LIN {X 0,Y 305.438,Z 295.055,A -85,B 0,C 180,E1 -15812.6,E2 -15812.6} C_VEL
LIN {X 0,Y 305.444,Z 295.06,A -85,B 0,C 180,E1 -15815.533,E2 -15815.533} C_VEL
LIN {X 0,Y 305.473,Z 295.058,A -85,B 0,C 180,E1 -15819.812,E2 -15819.812} C_VEL
LIN {X 0,Y 305.509,Z 295.056,A -85,B 0,C 180,E1 -15823.975,E2 -15823.975} C_VEL
LIN {X 0,Y 305.569,Z 295.038,A -85,B 0,C 180,E1 -15826.703,E2 -15826.703} C_VEL
LIN {X 0,Y 305.751,Z 295.012,A -85,B 0,C 180,E1 -15831.261,E2 -15831.261} C_VEL
LIN {X 0,Y 305.782,Z 295.02,A -85,B 0,C 180,E1 -15833.401,E2 -15833.401} C_VEL
LIN {X 0,Y 305.869,Z 295.005,A -85,B 0,C 180,E1 -15837.366,E2 -15837.366} C_VEL
LIN {X 0,Y 305.914,Z 294.996,A -85,B 0,C 180,E1 -15840,E2 -15840} C_VEL
LIN {X 0,Y 305.856,Z 295.009,A -85,B 0,C 180,E1 -15842.634,E2 -15842.634} C_VEL
LIN {X 0,Y 305.785,Z 295.01,A -85,B 0,C 180,E1 -15846.599,E2 -15846.599} C_VEL
LIN {X 0,Y 305.692,Z 295.03,A -85,B 0,C 180,E1 -15849.261,E2 -15849.261} C_VEL
LIN {X 0,Y 305.588,Z 295.045,A -85,B 0,C 180,E1 -15853.296,E2 -15853.296} C_VEL
LIN {X 0,Y 305.592,Z 295.037,A -85,B 0,C 180,E1 -15856.02,E2 -15856.02} C_VEL
LIN {X 0,Y 305.575,Z 295.039,A -85,B 0,C 180,E1 -15859.445,E2 -15859.445} C_VEL
LIN {X 0,Y 305.484,Z 295.047,A -85,B 0,C 180,E1 -15863.039,E2 -15863.039} C_VEL
LIN {X 0,Y 305.469,Z 295.029,A -85,B 0,C 180,E1 -15866.198,E2 -15866.198} C_VEL
LIN {X 0,Y 305.456,Z 295.061,A -85,B 0,C 180,E1 -15869.037,E2 -15869.037} C_VEL
LIN {X 0,Y 305.434,Z 295.035,A -85,B 0,C 180,E1 -15871.953,E2 -15871.953} C_VEL
LIN {X 0,Y 305.461,Z 295.061,A -85,B 0,C 180,E1 -15875.113,E2 -15875.113} C_VEL
LIN {X 0,Y 305.438,Z 295.047,A -85,B 0,C 180,E1 -15878.527,E2 -15878.527} C_VEL
LIN {X 0,Y 305.453,Z 295.061,A -85,B 0,C 180,E1 -15882.586,E2 -15882.586} C_VEL
LIN {X 0,Y 305.445,Z 295.147,A -85,B 0,C 180,E1 -15886.483,E2 -15886.483} C_VEL
LIN {X 0,Y 308.84,Z 306.244,A -85,B 0,C 180,E1 -15890.054,E2 -15890.054} C_VEL
LIN {X 0,Y 310.401,Z 311.623,A -85,B 0,C 180,E1 -15891.632,E2 -15891.632} C_VEL
LIN {X 0,Y 319.441,Z 329.134,A -85,B 0,C 180,E1 -15893.374,E2 -15893.374} C_VEL
LIN {X 0,Y 328.319,Z 348.755,A -85,B 0,C 180,E1 -15895.02,E2 -15895.02} C_VEL
LIN {X 0,Y 331.337,Z 366.984,A -85,B 0,C 180,E1 -15895.849,E2 -15895.849} C_VEL
LIN {X 0,Y 328.248,Z 458.224,A -85,B 0,C 180,E1 -15897.82,E2 -15897.82} C_VEL
LIN {X 0,Y 327.28,Z 480.74,A -85,B 0,C 180,E1 -15898.348,E2 -15898.348} C_VEL
LIN {X 0,Y 325.993,Z 496.154,A -85,B 0,C 180,E1 -15898.932,E2 -15898.932} C_VEL
LIN {X 0,Y 324.176,Z 511.053,A -85,B 0,C 180,E1 -15899.732,E2 -15899.732} C_VEL
LIN {X 0,Y 322.054,Z 525.725,A -85,B 0,C 180,E1 -15900.797,E2 -15900.797} C_VEL
LIN {X 0,Y 319.866,Z 538.691,A -85,B 0,C 180,E1 -15901.989,E2 -15901.989} C_VEL
LIN {X 0,Y 317.244,Z 552.138,A -85,B 0,C 180,E1 -15903.524,E2 -15903.524} C_VEL
LIN {X 0,Y 314.639,Z 564.393,A -85,B 0,C 180,E1 -15905.241,E2 -15905.241} C_VEL
LIN {X 0,Y 312.196,Z 575.594,A -85,B 0,C 180,E1 -15907.15,E2 -15907.15} C_VEL
LIN {X 0,Y 310.158,Z 585.029,A -85,B 0,C 180,E1 -15909.092,E2 -15909.092} C_VEL
LIN {X 0,Y 308.094,Z 594.317,A -85,B 0,C 180,E1 -15911.377,E2 -15911.377} C_VEL
LIN {X 0,Y 306.236,Z 603.068,A -85,B 0,C 180,E1 -15914.015,E2 -15914.015} C_VEL
LIN {X 0,Y 304.974,Z 610.103,A -85,B 0,C 180,E1 -15916.677,E2 -15916.677} C_VEL
LIN {X 0,Y 304.129,Z 615.64,A -85,B 0,C 180,E1 -15919.347,E2 -15919.347} C_VEL
LIN {X 0,Y 303.744,Z 619.836,A -85,B 0,C 180,E1 -15922.021,E2 -15922.021} C_VEL
LIN {X 0,Y 303.616,Z 622.781,A -85,B 0,C 180,E1 -15924.688,E2 -15924.688} C_VEL
LIN {X 0,Y 303.621,Z 624.54,A -85,B 0,C 180,E1 -15927.347,E2 -15927.347} C_VEL
LIN {X 0,Y 303.667,Z 625.142,A -85,B 0,C 180,E1 -15930.001,E2 -15930.001} C_VEL
LIN {X 0,Y 303.621,Z 624.53,A -85,B 0,C 180,E1 -15932.654,E2 -15932.654} C_VEL
LIN {X 0,Y 303.624,Z 622.559,A -85,B 0,C 180,E1 -15935.545,E2 -15935.545} C_VEL
LIN {X 0,Y 303.743,Z 619.805,A -85,B 0,C 180,E1 -15937.981,E2 -15937.981} C_VEL
LIN {X 0,Y 304.118,Z 615.604,A -85,B 0,C 180,E1 -15940.655,E2 -15940.655} C_VEL
LIN {X 0,Y 304.975,Z 610.051,A -85,B 0,C 180,E1 -15943.324,E2 -15943.324} C_VEL
LIN {X 0,Y 306.237,Z 602.995,A -85,B 0,C 180,E1 -15945.986,E2 -15945.986} C_VEL
LIN {X 0,Y 308.037,Z 594.228,A -85,B 0,C 180,E1 -15948.628,E2 -15948.628} C_VEL
LIN {X 0,Y 310.17,Z 584.929,A -85,B 0,C 180,E1 -15950.909,E2 -15950.909} C_VEL
LIN {X 0,Y 312.217,Z 575.478,A -85,B 0,C 180,E1 -15952.849,E2 -15952.849} C_VEL
LIN {X 0,Y 314.826,Z 563.229,A -85,B 0,C 180,E1 -15954.921,E2 -15954.921} C_VEL
LIN {X 0,Y 317.458,Z 550.75,A -85,B 0,C 180,E1 -15956.636,E2 -15956.636} C_VEL
LIN {X 0,Y 320.124,Z 536.95,A -85,B 0,C 180,E1 -15958.166,E2 -15958.166} C_VEL
LIN {X 0,Y 322.363,Z 523.433,A -85,B 0,C 180,E1 -15959.373,E2 -15959.373} C_VEL
LIN {X 0,Y 324.441,Z 508.338,A -85,B 0,C 180,E1 -15960.422,E2 -15960.422} C_VEL
LIN {X 0,Y 326.235,Z 493.273,A -85,B 0,C 180,E1 -15961.179,E2 -15961.179} C_VEL
LIN {X 0,Y 327.414,Z 477.475,A -85,B 0,C 180,E1 -15961.729,E2 -15961.729} C_VEL
LIN {X 0,Y 330.438,Z 392.663,A -85,B 0,C 180,E1 -15963.573,E2 -15963.573} C_VEL
LIN {X 0,Y 331.271,Z 366.999,A -85,B 0,C 180,E1 -15964.132,E2 -15964.132} C_VEL
LIN {X 0,Y 328.119,Z 348.323,A -85,B 0,C 180,E1 -15964.988,E2 -15964.988} C_VEL
LIN {X 0,Y 319.028,Z 328.324,A -85,B 0,C 180,E1 -15966.672,E2 -15966.672} C_VEL
LIN {X 0,Y 312.112,Z 315.044,A -85,B 0,C 180,E1 -15967.991,E2 -15967.991} C_VEL
LIN {X 0,Y 310.215,Z 311.17,A -85,B 0,C 180,E1 -15968.419,E2 -15968.419} C_VEL
LIN {X 0,Y 307.253,Z 301.008,A -85,B 0,C 180,E1 -15971.556,E2 -15971.556} C_VEL
LIN {X 0,Y 305.451,Z 295.059,A -85,B 0,C 180,E1 -15973.564,E2 -15973.564} C_VEL
LIN {X 0,Y 305.458,Z 295.049,A -85,B 0,C 180,E1 -15977.415,E2 -15977.415} C_VEL
LIN {X 0,Y 305.479,Z 295.055,A -85,B 0,C 180,E1 -15981.598,E2 -15981.598} C_VEL
LIN {X 0,Y 305.466,Z 295.052,A -85,B 0,C 180,E1 -15984.887,E2 -15984.887} C_VEL
LIN {X 0,Y 305.445,Z 295.056,A -85,B 0,C 180,E1 -15988.359,E2 -15988.359} C_VEL
LIN {X 0,Y 305.48,Z 295.05,A -85,B 0,C 180,E1 -15991.11,E2 -15991.11} C_VEL
LIN {X 0,Y 305.505,Z 295.046,A -85,B 0,C 180,E1 -15994.082,E2 -15994.082} C_VEL
LIN {X 0,Y 305.486,Z 295.055,A -85,B 0,C 180,E1 -15998.402,E2 -15998.402} C_VEL
LIN {X 0,Y 305.584,Z 295.036,A -85,B 0,C 180,E1 -16001.217,E2 -16001.217} C_VEL
LIN {X 0,Y 305.654,Z 295.029,A -85,B 0,C 180,E1 -16005.349,E2 -16005.349} C_VEL
LIN {X 0,Y 305.629,Z 295.031,A -85,B 0,C 180,E1 -16009.4,E2 -16009.4} C_VEL
LIN {X 0,Y 305.751,Z 295.018,A -85,B 0,C 180,E1 -16012.073,E2 -16012.073} C_VEL
LIN {X 0,Y 305.663,Z 295.035,A -85,B 0,C 180,E1 -16014.723,E2 -16014.723} C_VEL
LIN {X 0,Y 305.95,Z 294.998,A -85,B 0,C 180,E1 -16018.684,E2 -16018.684} C_VEL
LIN {X 0,Y 305.941,Z 294.993,A -85,B 0,C 180,E1 -16021.316,E2 -16021.316} C_VEL
LIN {X 0,Y 305.666,Z 295.03,A -85,B 0,C 180,E1 -16025.277,E2 -16025.277} C_VEL
LIN {X 0,Y 305.75,Z 295.026,A -85,B 0,C 180,E1 -16027.927,E2 -16027.927} C_VEL
LIN {X 0,Y 305.6,Z 295.042,A -85,B 0,C 180,E1 -16031.945,E2 -16031.945} C_VEL
LIN {X 0,Y 305.563,Z 295.038,A -85,B 0,C 180,E1 -16034.979,E2 -16034.979} C_VEL
LIN {X 0,Y 305.505,Z 295.046,A -85,B 0,C 180,E1 -16038.788,E2 -16038.788} C_VEL
LIN {X 0,Y 305.459,Z 295.053,A -85,B 0,C 180,E1 -16043.025,E2 -16043.025} C_VEL
LIN {X 0,Y 305.454,Z 295.052,A -85,B 0,C 180,E1 -16046.19,E2 -16046.19} C_VEL
LIN {X 0,Y 305.427,Z 295.039,A -85,B 0,C 180,E1 -16049.025,E2 -16049.025} C_VEL
LIN {X 0,Y 305.44,Z 295.061,A -85,B 0,C 180,E1 -16051.953,E2 -16051.953} C_VEL
LIN {X 0,Y 305.464,Z 295.059,A -85,B 0,C 180,E1 -16055.113,E2 -16055.113} C_VEL
LIN {X 0,Y 305.436,Z 295.058,A -85,B 0,C 180,E1 -16058.524,E2 -16058.524} C_VEL
LIN {X 0,Y 305.402,Z 295.066,A -85,B 0,C 180,E1 -16062.574,E2 -16062.574} C_VEL
LIN {X 0,Y 305.376,Z 295.066,A -85,B 0,C 180,E1 -16066.335,E2 -16066.335} C_VEL
LIN {X 0,Y 305.423,Z 295.064,A -85,B 0,C 180,E1 -16070.613,E2 -16070.613} C_VEL
LIN {X 0,Y 305.462,Z 295.277,A -85,B 0,C 180,E1 -16071.035,E2 -16071.035} C_VEL
LIN {X 0,Y 306.538,Z 298.105,A -85,B 0,C 180,E1 -16071.282,E2 -16071.282} C_VEL
LIN {X 0,Y 308.25,Z 300.361,A -85,B 0,C 180,E1 -16071.606,E2 -16071.606} C_VEL
LIN {X 0,Y 317.367,Z 315.01,A -85,B 0,C 180,E1 -16073.319,E2 -16073.319} C_VEL
LIN {X 0,Y 324.527,Z 328.876,A -85,B 0,C 180,E1 -16074.636,E2 -16074.636} C_VEL
LIN {X 0,Y 331.716,Z 344.391,A -85,B 0,C 180,E1 -16075.922,E2 -16075.922} C_VEL
LIN {X 0,Y 331.809,Z 349.272,A -85,B 0,C 180,E1 -16076.058,E2 -16076.058} C_VEL
LIN {X 0,Y 327.931,Z 457.659,A -85,B 0,C 180,E1 -16078.417,E2 -16078.417} C_VEL
LIN {X 0,Y 326.78,Z 473.515,A -85,B 0,C 180,E1 -16079.006,E2 -16079.006} C_VEL
LIN {X 0,Y 325.391,Z 488.142,A -85,B 0,C 180,E1 -16079.805,E2 -16079.805} C_VEL
LIN {X 0,Y 323.706,Z 501.433,A -85,B 0,C 180,E1 -16080.757,E2 -16080.757} C_VEL
LIN {X 0,Y 321.606,Z 514.984,A -85,B 0,C 180,E1 -16081.976,E2 -16081.976} C_VEL
LIN {X 0,Y 319.132,Z 528.731,A -85,B 0,C 180,E1 -16083.515,E2 -16083.515} C_VEL
LIN {X 0,Y 316.738,Z 540.07,A -85,B 0,C 180,E1 -16085.065,E2 -16085.065} C_VEL
LIN {X 0,Y 314.418,Z 551.5,A -85,B 0,C 180,E1 -16086.972,E2 -16086.972} C_VEL
LIN {X 0,Y 312.18,Z 561.12,A -85,B 0,C 180,E1 -16088.887,E2 -16088.887} C_VEL
LIN {X 0,Y 309.949,Z 570.544,A -85,B 0,C 180,E1 -16091.148,E2 -16091.148} C_VEL
LIN {X 0,Y 307.923,Z 579.033,A -85,B 0,C 180,E1 -16093.644,E2 -16093.644} C_VEL
LIN {X 0,Y 306.53,Z 585.692,A -85,B 0,C 180,E1 -16096.069,E2 -16096.069} C_VEL
LIN {X 0,Y 305.314,Z 591.489,A -85,B 0,C 180,E1 -16098.716,E2 -16098.716} C_VEL
LIN {X 0,Y 304.655,Z 594.918,A -85,B 0,C 180,E1 -16100.706,E2 -16100.706} C_VEL
LIN {X 0,Y 304.077,Z 598.682,A -85,B 0,C 180,E1 -16103.639,E2 -16103.639} C_VEL
LIN {X 0,Y 303.861,Z 600.677,A -85,B 0,C 180,E1 -16106.021,E2 -16106.021} C_VEL
LIN {X 0,Y 303.676,Z 601.848,A -85,B 0,C 180,E1 -16108.673,E2 -16108.673} C_VEL
LIN {X 0,Y 303.676,Z 601.862,A -85,B 0,C 180,E1 -16111.325,E2 -16111.325} C_VEL
LIN {X 0,Y 303.86,Z 600.747,A -85,B 0,C 180,E1 -16113.978,E2 -16113.978} C_VEL
LIN {X 0,Y 304.127,Z 598.511,A -85,B 0,C 180,E1 -16116.634,E2 -16116.634} C_VEL
LIN {X 0,Y 304.649,Z 595.093,A -85,B 0,C 180,E1 -16119.292,E2 -16119.292} C_VEL
LIN {X 0,Y 305.52,Z 590.409,A -85,B 0,C 180,E1 -16121.948,E2 -16121.948} C_VEL
LIN {X 0,Y 306.853,Z 584.331,A -85,B 0,C 180,E1 -16124.592,E2 -16124.592} C_VEL
LIN {X 0,Y 308.526,Z 576.675,A -85,B 0,C 180,E1 -16127.225,E2 -16127.225} C_VEL
LIN {X 0,Y 310.464,Z 568.504,A -85,B 0,C 180,E1 -16129.505,E2 -16129.505} C_VEL
LIN {X 0,Y 312.774,Z 558.653,A -85,B 0,C 180,E1 -16131.762,E2 -16131.762} C_VEL
LIN {X 0,Y 315.063,Z 548.548,A -85,B 0,C 180,E1 -16133.673,E2 -16133.673} C_VEL
LIN {X 0,Y 317.528,Z 536.513,A -85,B 0,C 180,E1 -16135.569,E2 -16135.569} C_VEL
LIN {X 0,Y 319.998,Z 524.429,A -85,B 0,C 180,E1 -16137.111,E2 -16137.111} C_VEL
LIN {X 0,Y 322.274,Z 511.296,A -85,B 0,C 180,E1 -16138.492,E2 -16138.492} C_VEL
LIN {X 0,Y 324.071,Z 498.775,A -85,B 0,C 180,E1 -16139.562,E2 -16139.562} C_VEL
LIN {X 0,Y 325.751,Z 484.936,A -85,B 0,C 180,E1 -16140.497,E2 -16140.497} C_VEL
LIN {X 0,Y 327.156,Z 469.761,A -85,B 0,C 180,E1 -16141.26,E2 -16141.26} C_VEL
LIN {X 0,Y 328.161,Z 454.114,A -85,B 0,C 180,E1 -16141.783,E2 -16141.783} C_VEL
LIN {X 0,Y 331.159,Z 369.826,A -85,B 0,C 180,E1 -16143.608,E2 -16143.608} C_VEL
LIN {X 0,Y 330.87,Z 364.028,A -85,B 0,C 180,E1 -16143.79,E2 -16143.79} C_VEL
LIN {X 0,Y 329.712,Z 358.441,A -85,B 0,C 180,E1 -16144.071,E2 -16144.071} C_VEL
LIN {X 0,Y 325.964,Z 347.786,A -85,B 0,C 180,E1 -16144.802,E2 -16144.802} C_VEL
LIN {X 0,Y 323.29,Z 340.745,A -85,B 0,C 180,E1 -16145.323,E2 -16145.323} C_VEL
LIN {X 0,Y 314.907,Z 323.642,A -85,B 0,C 180,E1 -16146.899,E2 -16146.899} C_VEL
LIN {X 0,Y 308.972,Z 313.39,A -85,B 0,C 180,E1 -16148.034,E2 -16148.034} C_VEL
LIN {X 0,Y 302.699,Z 303.653,A -85,B 0,C 180,E1 -16149.27,E2 -16149.27} C_VEL
LIN {X 0,Y 300.712,Z 300.374,A -85,B 0,C 180,E1 -16149.683,E2 -16149.683} C_VEL
LIN {X 0,Y 298.917,Z 297.892,A -85,B 0,C 180,E1 -16150.048,E2 -16150.048} C_VEL
LIN {X 0,Y 298.38,Z 295.941,A -85,B 0,C 180,E1 -16150.218,E2 -16150.218} C_VEL
LIN {X 0,Y 298.367,Z 295.926,A -85,B 0,C 180,E1 -16153.097,E2 -16153.097} C_VEL
LIN {X 0,Y 298.367,Z 295.925,A -85,B 0,C 180,E1 -16156.914,E2 -16156.914} C_VEL
LIN {X 0,Y 298.352,Z 295.945,A -85,B 0,C 180,E1 -16161.018,E2 -16161.018} C_VEL
LIN {X 0,Y 298.401,Z 295.908,A -85,B 0,C 180,E1 -16163.928,E2 -16163.928} C_VEL
LIN {X 0,Y 298.39,Z 295.941,A -85,B 0,C 180,E1 -16167.199,E2 -16167.199} C_VEL
LIN {X 0,Y 298.361,Z 295.947,A -85,B 0,C 180,E1 -16170.638,E2 -16170.638} C_VEL
LIN {X 0,Y 298.414,Z 295.938,A -85,B 0,C 180,E1 -16174.917,E2 -16174.917} C_VEL
LIN {X 0,Y 298.388,Z 295.936,A -85,B 0,C 180,E1 -16177.861,E2 -16177.861} C_VEL
LIN {X 0,Y 298.45,Z 295.922,A -85,B 0,C 180,E1 -16180.751,E2 -16180.751} C_VEL
LIN {X 0,Y 298.508,Z 295.919,A -85,B 0,C 180,E1 -16184.99,E2 -16184.99} C_VEL
LIN {X 0,Y 298.58,Z 295.915,A -85,B 0,C 180,E1 -16189.146,E2 -16189.146} C_VEL
LIN {X 0,Y 298.695,Z 295.894,A -85,B 0,C 180,E1 -16191.884,E2 -16191.884} C_VEL
LIN {X 0,Y 298.629,Z 295.905,A -85,B 0,C 180,E1 -16194.598,E2 -16194.598} C_VEL
LIN {X 0,Y 298.905,Z 295.877,A -85,B 0,C 180,E1 -16198.653,E2 -16198.653} C_VEL
LIN {X 0,Y 298.912,Z 295.862,A -85,B 0,C 180,E1 -16201.347,E2 -16201.347} C_VEL
LIN {X 0,Y 298.734,Z 295.89,A -85,B 0,C 180,E1 -16206.755,E2 -16206.755} C_VEL
LIN {X 0,Y 298.624,Z 295.909,A -85,B 0,C 180,E1 -16209.482,E2 -16209.482} C_VEL
LIN {X 0,Y 298.551,Z 295.923,A -85,B 0,C 180,E1 -16213.615,E2 -16213.615} C_VEL
LIN {X 0,Y 298.547,Z 295.919,A -85,B 0,C 180,E1 -16216.409,E2 -16216.409} C_VEL
LIN {X 0,Y 298.509,Z 295.919,A -85,B 0,C 180,E1 -16219.655,E2 -16219.655} C_VEL
LIN {X 0,Y 298.422,Z 295.916,A -85,B 0,C 180,E1 -16223.601,E2 -16223.601} C_VEL
LIN {X 0,Y 298.408,Z 295.913,A -85,B 0,C 180,E1 -16226.582,E2 -16226.582} C_VEL
LIN {X 0,Y 298.395,Z 295.935,A -85,B 0,C 180,E1 -16229.644,E2 -16229.644} C_VEL
LIN {X 0,Y 298.39,Z 295.916,A -85,B 0,C 180,E1 -16232.801,E2 -16232.801} C_VEL
LIN {X 0,Y 298.442,Z 295.915,A -85,B 0,C 180,E1 -16236.807,E2 -16236.807} C_VEL
LIN {X 0,Y 298.385,Z 295.939,A -85,B 0,C 180,E1 -16241.088,E2 -16241.088} C_VEL
LIN {X 0,Y 298.396,Z 295.938,A -85,B 0,C 180,E1 -16243.104,E2 -16243.104} C_VEL
LIN {X 0,Y 298.373,Z 296.083,A -85,B 0,C 180,E1 -16245.56,E2 -16245.56} C_VEL
LIN {X 0,Y 301.47,Z 305.891,A -85,B 0,C 180,E1 -16248.871,E2 -16248.871} C_VEL
LIN {X 0,Y 303.07,Z 311.245,A -85,B 0,C 180,E1 -16250.525,E2 -16250.525} C_VEL
LIN {X 0,Y 311.578,Z 327.368,A -85,B 0,C 180,E1 -16252.251,E2 -16252.251} C_VEL
LIN {X 0,Y 318.889,Z 342.773,A -85,B 0,C 180,E1 -16253.674,E2 -16253.674} C_VEL
LIN {X 0,Y 322.894,Z 352.057,A -85,B 0,C 180,E1 -16254.438,E2 -16254.438} C_VEL
LIN {X 0,Y 325.461,Z 368.965,A -85,B 0,C 180,E1 -16255.203,E2 -16255.203} C_VEL
LIN {X 0,Y 321.698,Z 472.084,A -85,B 0,C 180,E1 -16257.455,E2 -16257.455} C_VEL
LIN {X 0,Y 320.687,Z 488.035,A -85,B 0,C 180,E1 -16257.943,E2 -16257.943} C_VEL
LIN {X 0,Y 319.067,Z 503.234,A -85,B 0,C 180,E1 -16258.643,E2 -16258.643} C_VEL
LIN {X 0,Y 317.13,Z 517.416,A -85,B 0,C 180,E1 -16259.538,E2 -16259.538} C_VEL
LIN {X 0,Y 314.742,Z 532.154,A -85,B 0,C 180,E1 -16260.761,E2 -16260.761} C_VEL
LIN {X 0,Y 312.172,Z 545.471,A -85,B 0,C 180,E1 -16262.151,E2 -16262.151} C_VEL
LIN {X 0,Y 309.591,Z 557.73,A -85,B 0,C 180,E1 -16263.726,E2 -16263.726} C_VEL
LIN {X 0,Y 306.808,Z 569.962,A -85,B 0,C 180,E1 -16265.65,E2 -16265.65} C_VEL
LIN {X 0,Y 304.278,Z 580.95,A -85,B 0,C 180,E1 -16267.762,E2 -16267.762} C_VEL
LIN {X 0,Y 302.135,Z 590.295,A -85,B 0,C 180,E1 -16269.935,E2 -16269.935} C_VEL
LIN {X 0,Y 300.219,Z 598.651,A -85,B 0,C 180,E1 -16272.283,E2 -16272.283} C_VEL
LIN {X 0,Y 298.585,Z 606.512,A -85,B 0,C 180,E1 -16274.995,E2 -16274.995} C_VEL
LIN {X 0,Y 297.523,Z 612.777,A -85,B 0,C 180,E1 -16277.726,E2 -16277.726} C_VEL
LIN {X 0,Y 296.853,Z 617.628,A -85,B 0,C 180,E1 -16280.461,E2 -16280.461} C_VEL
LIN {X 0,Y 296.61,Z 621.191,A -85,B 0,C 180,E1 -16283.197,E2 -16283.197} C_VEL
LIN {X 0,Y 296.515,Z 623.535,A -85,B 0,C 180,E1 -16285.923,E2 -16285.923} C_VEL
LIN {X 0,Y 296.539,Z 624.715,A -85,B 0,C 180,E1 -16288.643,E2 -16288.643} C_VEL
LIN {X 0,Y 296.58,Z 624.872,A -85,B 0,C 180,E1 -16290.001,E2 -16290.001} C_VEL
LIN {X 0,Y 296.545,Z 624.26,A -85,B 0,C 180,E1 -16292.717,E2 -16292.717} C_VEL
LIN {X 0,Y 296.545,Z 622.43,A -85,B 0,C 180,E1 -16295.509,E2 -16295.509} C_VEL
LIN {X 0,Y 296.671,Z 619.532,A -85,B 0,C 180,E1 -16298.172,E2 -16298.172} C_VEL
LIN {X 0,Y 297.081,Z 615.33,A -85,B 0,C 180,E1 -16300.91,E2 -16300.91} C_VEL
LIN {X 0,Y 297.991,Z 609.776,A -85,B 0,C 180,E1 -16303.642,E2 -16303.642} C_VEL
LIN {X 0,Y 299.338,Z 602.72,A -85,B 0,C 180,E1 -16306.365,E2 -16306.365} C_VEL
LIN {X 0,Y 301.22,Z 593.952,A -85,B 0,C 180,E1 -16309.066,E2 -16309.066} C_VEL
LIN {X 0,Y 303.47,Z 584.653,A -85,B 0,C 180,E1 -16311.393,E2 -16311.393} C_VEL
LIN {X 0,Y 305.619,Z 575.203,A -85,B 0,C 180,E1 -16313.372,E2 -16313.372} C_VEL
LIN {X 0,Y 308.359,Z 562.954,A -85,B 0,C 180,E1 -16315.481,E2 -16315.481} C_VEL
LIN {X 0,Y 311.11,Z 550.475,A -85,B 0,C 180,E1 -16317.223,E2 -16317.223} C_VEL
LIN {X 0,Y 313.844,Z 536.673,A -85,B 0,C 180,E1 -16318.781,E2 -16318.781} C_VEL
LIN {X 0,Y 316.226,Z 522.786,A -85,B 0,C 180,E1 -16320.035,E2 -16320.035} C_VEL
LIN {X 0,Y 318.34,Z 508.06,A -85,B 0,C 180,E1 -16321.068,E2 -16321.068} C_VEL
LIN {X 0,Y 320.162,Z 492.991,A -85,B 0,C 180,E1 -16321.839,E2 -16321.839} C_VEL
LIN {X 0,Y 321.391,Z 477.186,A -85,B 0,C 180,E1 -16322.396,E2 -16322.396} C_VEL
LIN {X 0,Y 324.541,Z 392.371,A -85,B 0,C 180,E1 -16324.267,E2 -16324.267} C_VEL
LIN {X 0,Y 325.32,Z 367.579,A -85,B 0,C 180,E1 -16324.823,E2 -16324.823} C_VEL
LIN {X 0,Y 322.434,Z 350.858,A -85,B 0,C 180,E1 -16325.622,E2 -16325.622} C_VEL
LIN {X 0,Y 313.668,Z 331.535,A -85,B 0,C 180,E1 -16327.306,E2 -16327.306} C_VEL
LIN {X 0,Y 307.392,Z 319.423,A -85,B 0,C 180,E1 -16328.546,E2 -16328.546} C_VEL
LIN {X 0,Y 302.907,Z 310.838,A -85,B 0,C 180,E1 -16329.518,E2 -16329.518} C_VEL
LIN {X 0,Y 299.879,Z 300.642,A -85,B 0,C 180,E1 -16332.817,E2 -16332.817} C_VEL
LIN {X 0,Y 298.373,Z 295.945,A -85,B 0,C 180,E1 -16334.485,E2 -16334.485} C_VEL
LIN {X 0,Y 298.406,Z 295.924,A -85,B 0,C 180,E1 -16336.921,E2 -16336.921} C_VEL
LIN {X 0,Y 298.407,Z 295.939,A -85,B 0,C 180,E1 -16341.007,E2 -16341.007} C_VEL
LIN {X 0,Y 298.422,Z 295.934,A -85,B 0,C 180,E1 -16343.931,E2 -16343.931} C_VEL
LIN {X 0,Y 298.392,Z 295.932,A -85,B 0,C 180,E1 -16347.986,E2 -16347.986} C_VEL
LIN {X 0,Y 298.418,Z 295.933,A -85,B 0,C 180,E1 -16351.9,E2 -16351.9} C_VEL
LIN {X 0,Y 298.449,Z 295.93,A -85,B 0,C 180,E1 -16354.921,E2 -16354.921} C_VEL
LIN {X 0,Y 298.442,Z 295.934,A -85,B 0,C 180,E1 -16359.315,E2 -16359.315} C_VEL
LIN {X 0,Y 298.539,Z 295.921,A -85,B 0,C 180,E1 -16362.18,E2 -16362.18} C_VEL
LIN {X 0,Y 298.598,Z 295.907,A -85,B 0,C 180,E1 -16364.995,E2 -16364.995} C_VEL
LIN {X 0,Y 298.588,Z 295.907,A -85,B 0,C 180,E1 -16369.147,E2 -16369.147} C_VEL
LIN {X 0,Y 298.702,Z 295.898,A -85,B 0,C 180,E1 -16371.885,E2 -16371.885} C_VEL
LIN {X 0,Y 298.633,Z 295.911,A -85,B 0,C 180,E1 -16374.599,E2 -16374.599} C_VEL
LIN {X 0,Y 298.917,Z 295.874,A -85,B 0,C 180,E1 -16378.653,E2 -16378.653} C_VEL
LIN {X 0,Y 298.909,Z 295.868,A -85,B 0,C 180,E1 -16381.347,E2 -16381.347} C_VEL
LIN {X 0,Y 298.738,Z 295.891,A -85,B 0,C 180,E1 -16386.755,E2 -16386.755} C_VEL
LIN {X 0,Y 298.63,Z 295.907,A -85,B 0,C 180,E1 -16389.482,E2 -16389.482} C_VEL
LIN {X 0,Y 298.528,Z 295.92,A -85,B 0,C 180,E1 -16393.617,E2 -16393.617} C_VEL
LIN {X 0,Y 298.456,Z 295.933,A -85,B 0,C 180,E1 -16396.414,E2 -16396.414} C_VEL
LIN {X 0,Y 298.435,Z 295.93,A -85,B 0,C 180,E1 -16399.611,E2 -16399.611} C_VEL
LIN {X 0,Y 298.392,Z 295.937,A -85,B 0,C 180,E1 -16403.603,E2 -16403.603} C_VEL
LIN {X 0,Y 298.405,Z 295.921,A -85,B 0,C 180,E1 -16406.583,E2 -16406.583} C_VEL
LIN {X 0,Y 298.36,Z 295.927,A -85,B 0,C 180,E1 -16409.648,E2 -16409.648} C_VEL
LIN {X 0,Y 298.396,Z 295.935,A -85,B 0,C 180,E1 -16412.8,E2 -16412.8} C_VEL
LIN {X 0,Y 298.429,Z 295.932,A -85,B 0,C 180,E1 -16416.802,E2 -16416.802} C_VEL
LIN {X 0,Y 298.375,Z 295.939,A -85,B 0,C 180,E1 -16419.492,E2 -16419.492} C_VEL
LIN {X 0,Y 298.369,Z 295.942,A -85,B 0,C 180,E1 -16423.096,E2 -16423.096} C_VEL
LIN {X 0,Y 298.342,Z 295.946,A -85,B 0,C 180,E1 -16426.909,E2 -16426.909} C_VEL
LIN {X 0,Y 298.357,Z 295.961,A -85,B 0,C 180,E1 -16429.932,E2 -16429.932} C_VEL
LIN {X 0,Y 299.222,Z 298.569,A -85,B 0,C 180,E1 -16430.153,E2 -16430.153} C_VEL
LIN {X 0,Y 301.208,Z 301.162,A -85,B 0,C 180,E1 -16430.549,E2 -16430.549} C_VEL
LIN {X 0,Y 309.354,Z 313.972,A -85,B 0,C 180,E1 -16432.164,E2 -16432.164} C_VEL
LIN {X 0,Y 314.579,Z 323.063,A -85,B 0,C 180,E1 -16433.162,E2 -16433.162} C_VEL
LIN {X 0,Y 323.863,Z 342.042,A -85,B 0,C 180,E1 -16434.903,E2 -16434.903} C_VEL
LIN {X 0,Y 325.948,Z 346.833,A -85,B 0,C 180,E1 -16435.29,E2 -16435.29} C_VEL
LIN {X 0,Y 323.412,Z 419.399,A -85,B 0,C 180,E1 -16436.886,E2 -16436.886} C_VEL
LIN {X 0,Y 321.926,Z 457.946,A -85,B 0,C 180,E1 -16437.757,E2 -16437.757} C_VEL
LIN {X 0,Y 320.715,Z 473.847,A -85,B 0,C 180,E1 -16438.356,E2 -16438.356} C_VEL
LIN {X 0,Y 319.373,Z 487.649,A -85,B 0,C 180,E1 -16439.118,E2 -16439.118} C_VEL
LIN {X 0,Y 317.535,Z 501.71,A -85,B 0,C 180,E1 -16440.132,E2 -16440.132} C_VEL
LIN {X 0,Y 315.374,Z 515.259,A -85,B 0,C 180,E1 -16441.371,E2 -16441.371} C_VEL
LIN {X 0,Y 313.034,Z 527.721,A -85,B 0,C 180,E1 -16442.777,E2 -16442.777} C_VEL
LIN {X 0,Y 310.518,Z 539.283,A -85,B 0,C 180,E1 -16444.35,E2 -16444.35} C_VEL
LIN {X 0,Y 308.277,Z 550.006,A -85,B 0,C 180,E1 -16446.13,E2 -16446.13} C_VEL
LIN {X 0,Y 305.873,Z 559.923,A -85,B 0,C 180,E1 -16448.075,E2 -16448.075} C_VEL
LIN {X 0,Y 303.534,Z 569.598,A -85,B 0,C 180,E1 -16450.382,E2 -16450.382} C_VEL
LIN {X 0,Y 301.51,Z 577.663,A -85,B 0,C 180,E1 -16452.711,E2 -16452.711} C_VEL
LIN {X 0,Y 300.026,Z 584.3,A -85,B 0,C 180,E1 -16455.067,E2 -16455.067} C_VEL
LIN {X 0,Y 298.586,Z 590.449,A -85,B 0,C 180,E1 -16457.769,E2 -16457.769} C_VEL
LIN {X 0,Y 297.644,Z 595.189,A -85,B 0,C 180,E1 -16460.486,E2 -16460.486} C_VEL
LIN {X 0,Y 297.009,Z 599.105,A -85,B 0,C 180,E1 -16463.632,E2 -16463.632} C_VEL
LIN {X 0,Y 296.799,Z 600.947,A -85,B 0,C 180,E1 -16465.926,E2 -16465.926} C_VEL
LIN {X 0,Y 296.592,Z 602.118,A -85,B 0,C 180,E1 -16468.642,E2 -16468.642} C_VEL
LIN {X 0,Y 296.592,Z 602.132,A -85,B 0,C 180,E1 -16471.357,E2 -16471.357} C_VEL
LIN {X 0,Y 296.798,Z 601.017,A -85,B 0,C 180,E1 -16474.073,E2 -16474.073} C_VEL
LIN {X 0,Y 297.065,Z 598.782,A -85,B 0,C 180,E1 -16476.793,E2 -16476.793} C_VEL
LIN {X 0,Y 297.637,Z 595.363,A -85,B 0,C 180,E1 -16479.513,E2 -16479.513} C_VEL
LIN {X 0,Y 298.555,Z 590.679,A -85,B 0,C 180,E1 -16482.231,E2 -16482.231} C_VEL
LIN {X 0,Y 299.955,Z 584.601,A -85,B 0,C 180,E1 -16484.935,E2 -16484.935} C_VEL
LIN {X 0,Y 301.707,Z 576.946,A -85,B 0,C 180,E1 -16487.627,E2 -16487.627} C_VEL
LIN {X 0,Y 303.756,Z 568.773,A -85,B 0,C 180,E1 -16489.954,E2 -16489.954} C_VEL
LIN {X 0,Y 306.16,Z 558.922,A -85,B 0,C 180,E1 -16492.256,E2 -16492.256} C_VEL
LIN {X 0,Y 308.532,Z 548.817,A -85,B 0,C 180,E1 -16494.205,E2 -16494.205} C_VEL
LIN {X 0,Y 311.151,Z 536.779,A -85,B 0,C 180,E1 -16496.132,E2 -16496.132} C_VEL
LIN {X 0,Y 313.69,Z 524.695,A -85,B 0,C 180,E1 -16497.702,E2 -16497.702} C_VEL
LIN {X 0,Y 316.055,Z 511.561,A -85,B 0,C 180,E1 -16499.105,E2 -16499.105} C_VEL
LIN {X 0,Y 317.92,Z 499.039,A -85,B 0,C 180,E1 -16500.193,E2 -16500.193} C_VEL
LIN {X 0,Y 319.76,Z 484.379,A -85,B 0,C 180,E1 -16501.189,E2 -16501.189} C_VEL
LIN {X 0,Y 321.184,Z 469.106,A -85,B 0,C 180,E1 -16501.955,E2 -16501.955} C_VEL
LIN {X 0,Y 322.16,Z 454.364,A -85,B 0,C 180,E1 -16502.446,E2 -16502.446} C_VEL
LIN {X 0,Y 326.137,Z 348.068,A -85,B 0,C 180,E1 -16504.773,E2 -16504.773} C_VEL
LIN {X 0,Y 325.775,Z 346.371,A -85,B 0,C 180,E1 -16504.863,E2 -16504.863} C_VEL
LIN {X 0,Y 323.29,Z 340.745,A -85,B 0,C 180,E1 -16505.323,E2 -16505.323} C_VEL
LIN {X 0,Y 321.772,Z 337.507,A -85,B 0,C 180,E1 -16505.604,E2 -16505.604} C_VEL
LIN {X 0,Y 319.783,Z 334.691,A -85,B 0,C 180,E1 -16505.939,E2 -16505.939} C_VEL
LIN {X 0,Y 315.041,Z 329.938,A -85,B 0,C 180,E1 -16506.705,E2 -16506.705} C_VEL
LIN {X 0,Y 310.03,Z 325.446,A -85,B 0,C 180,E1 -16507.533,E2 -16507.533} C_VEL
LIN {X 0,Y 306.694,Z 321.584,A -85,B 0,C 180,E1 -16508.131,E2 -16508.131} C_VEL
LIN {X 0,Y 305.744,Z 320.112,A -85,B 0,C 180,E1 -16508.315,E2 -16508.315} C_VEL
LIN {X 0,Y 296.298,Z 305.289,A -85,B 0,C 180,E1 -16510.248,E2 -16510.248} C_VEL
LIN {X 0,Y 293.477,Z 301.11,A -85,B 0,C 180,E1 -16510.852,E2 -16510.852} C_VEL
LIN {X 0,Y 291.766,Z 298.605,A -85,B 0,C 180,E1 -16511.227,E2 -16511.227} C_VEL
LIN {X 0,Y 291.313,Z 296.822,A -85,B 0,C 180,E1 -16511.385,E2 -16511.385} C_VEL
LIN {X 0,Y 291.28,Z 296.828,A -85,B 0,C 180,E1 -16515.596,E2 -16515.596} C_VEL
LIN {X 0,Y 291.292,Z 296.811,A -85,B 0,C 180,E1 -16519.35,E2 -16519.35} C_VEL
LIN {X 0,Y 291.383,Z 296.785,A -85,B 0,C 180,E1 -16522.916,E2 -16522.916} C_VEL
LIN {X 0,Y 291.341,Z 296.816,A -85,B 0,C 180,E1 -16526.301,E2 -16526.301} C_VEL
LIN {X 0,Y 291.332,Z 296.82,A -85,B 0,C 180,E1 -16530.278,E2 -16530.278} C_VEL
LIN {X 0,Y 291.341,Z 296.819,A -85,B 0,C 180,E1 -16534.265,E2 -16534.265} C_VEL
LIN {X 0,Y 291.347,Z 296.81,A -85,B 0,C 180,E1 -16537.297,E2 -16537.297} C_VEL
LIN {X 0,Y 291.382,Z 296.806,A -85,B 0,C 180,E1 -16540.265,E2 -16540.265} C_VEL
LIN {X 0,Y 291.472,Z 296.797,A -85,B 0,C 180,E1 -16544.682,E2 -16544.682} C_VEL
LIN {X 0,Y 291.525,Z 296.795,A -85,B 0,C 180,E1 -16548.88,E2 -16548.88} C_VEL
LIN {X 0,Y 291.649,Z 296.771,A -85,B 0,C 180,E1 -16551.687,E2 -16551.687} C_VEL
LIN {X 0,Y 291.598,Z 296.782,A -85,B 0,C 180,E1 -16554.468,E2 -16554.468} C_VEL
LIN {X 0,Y 291.872,Z 296.753,A -85,B 0,C 180,E1 -16558.62,E2 -16558.62} C_VEL
LIN {X 0,Y 291.878,Z 296.738,A -85,B 0,C 180,E1 -16561.38,E2 -16561.38} C_VEL
LIN {X 0,Y 291.686,Z 296.768,A -85,B 0,C 180,E1 -16566.919,E2 -16566.919} C_VEL
LIN {X 0,Y 291.566,Z 296.785,A -85,B 0,C 180,E1 -16569.714,E2 -16569.714} C_VEL
LIN {X 0,Y 291.521,Z 296.794,A -85,B 0,C 180,E1 -16573.95,E2 -16573.95} C_VEL
LIN {X 0,Y 291.485,Z 296.802,A -85,B 0,C 180,E1 -16576.818,E2 -16576.818} C_VEL
LIN {X 0,Y 291.449,Z 296.799,A -85,B 0,C 180,E1 -16579.875,E2 -16579.875} C_VEL
LIN {X 0,Y 291.362,Z 296.786,A -85,B 0,C 180,E1 -16584.208,E2 -16584.208} C_VEL
LIN {X 0,Y 291.355,Z 296.803,A -85,B 0,C 180,E1 -16587.278,E2 -16587.278} C_VEL
LIN {X 0,Y 291.318,Z 296.805,A -85,B 0,C 180,E1 -16590.439,E2 -16590.439} C_VEL
LIN {X 0,Y 291.342,Z 296.807,A -85,B 0,C 180,E1 -16593.699,E2 -16593.699} C_VEL
LIN {X 0,Y 291.37,Z 296.793,A -85,B 0,C 180,E1 -16597.253,E2 -16597.253} C_VEL
LIN {X 0,Y 291.33,Z 296.819,A -85,B 0,C 180,E1 -16600.643,E2 -16600.643} C_VEL
LIN {X 0,Y 291.31,Z 296.875,A -85,B 0,C 180,E1 -16604.534,E2 -16604.534} C_VEL
LIN {X 0,Y 294.487,Z 306.922,A -85,B 0,C 180,E1 -16608.07,E2 -16608.07} C_VEL
LIN {X 0,Y 295.654,Z 310.793,A -85,B 0,C 180,E1 -16609.327,E2 -16609.327} C_VEL
LIN {X 0,Y 298.276,Z 315.425,A -85,B 0,C 180,E1 -16609.897,E2 -16609.897} C_VEL
LIN {X 0,Y 306.259,Z 330.532,A -85,B 0,C 180,E1 -16611.576,E2 -16611.576} C_VEL
LIN {X 0,Y 313.591,Z 346.083,A -85,B 0,C 180,E1 -16613.058,E2 -16613.058} C_VEL
LIN {X 0,Y 317.388,Z 355.144,A -85,B 0,C 180,E1 -16613.816,E2 -16613.816} C_VEL
LIN {X 0,Y 319.616,Z 370.103,A -85,B 0,C 180,E1 -16614.509,E2 -16614.509} C_VEL
LIN {X 0,Y 315.451,Z 477.851,A -85,B 0,C 180,E1 -16616.919,E2 -16616.919} C_VEL
LIN {X 0,Y 314.211,Z 493.273,A -85,B 0,C 180,E1 -16617.486,E2 -16617.486} C_VEL
LIN {X 0,Y 312.323,Z 508.183,A -85,B 0,C 180,E1 -16618.266,E2 -16618.266} C_VEL
LIN {X 0,Y 310.074,Z 523.165,A -85,B 0,C 180,E1 -16619.339,E2 -16619.339} C_VEL
LIN {X 0,Y 307.648,Z 536.647,A -85,B 0,C 180,E1 -16620.584,E2 -16620.584} C_VEL
LIN {X 0,Y 305.095,Z 549.094,A -85,B 0,C 180,E1 -16622.009,E2 -16622.009} C_VEL
LIN {X 0,Y 302.216,Z 561.763,A -85,B 0,C 180,E1 -16623.779,E2 -16623.779} C_VEL
LIN {X 0,Y 299.446,Z 573.282,A -85,B 0,C 180,E1 -16625.75,E2 -16625.75} C_VEL
LIN {X 0,Y 297.078,Z 582.987,A -85,B 0,C 180,E1 -16627.759,E2 -16627.759} C_VEL
LIN {X 0,Y 294.768,Z 592.528,A -85,B 0,C 180,E1 -16630.139,E2 -16630.139} C_VEL
LIN {X 0,Y 292.888,Z 600.485,A -85,B 0,C 180,E1 -16632.546,E2 -16632.546} C_VEL
LIN {X 0,Y 291.331,Z 607.925,A -85,B 0,C 180,E1 -16635.328,E2 -16635.328} C_VEL
LIN {X 0,Y 290.281,Z 613.836,A -85,B 0,C 180,E1 -16638.125,E2 -16638.125} C_VEL
LIN {X 0,Y 289.782,Z 617.355,A -85,B 0,C 180,E1 -16640.226,E2 -16640.226} C_VEL
LIN {X 0,Y 289.533,Z 620.92,A -85,B 0,C 180,E1 -16643.03,E2 -16643.03} C_VEL
LIN {X 0,Y 289.418,Z 623.265,A -85,B 0,C 180,E1 -16645.823,E2 -16645.823} C_VEL
LIN {X 0,Y 289.457,Z 624.446,A -85,B 0,C 180,E1 -16648.609,E2 -16648.609} C_VEL
LIN {X 0,Y 289.457,Z 624.442,A -85,B 0,C 180,E1 -16651.392,E2 -16651.392} C_VEL
LIN {X 0,Y 289.418,Z 623.247,A -85,B 0,C 180,E1 -16654.178,E2 -16654.178} C_VEL
LIN {X 0,Y 289.485,Z 620.888,A -85,B 0,C 180,E1 -16656.973,E2 -16656.973} C_VEL
LIN {X 0,Y 289.779,Z 617.319,A -85,B 0,C 180,E1 -16659.775,E2 -16659.775} C_VEL
LIN {X 0,Y 290.52,Z 612.458,A -85,B 0,C 180,E1 -16662.576,E2 -16662.576} C_VEL
LIN {X 0,Y 291.693,Z 605.902,A -85,B 0,C 180,E1 -16665.475,E2 -16665.475} C_VEL
LIN {X 0,Y 293.374,Z 598.291,A -85,B 0,C 180,E1 -16668.146,E2 -16668.146} C_VEL
LIN {X 0,Y 295.406,Z 589.924,A -85,B 0,C 180,E1 -16670.544,E2 -16670.544} C_VEL
LIN {X 0,Y 297.772,Z 580.095,A -85,B 0,C 180,E1 -16672.864,E2 -16672.864} C_VEL
LIN {X 0,Y 300.287,Z 569.558,A -85,B 0,C 180,E1 -16674.916,E2 -16674.916} C_VEL
LIN {X 0,Y 303.181,Z 557.303,A -85,B 0,C 180,E1 -16676.875,E2 -16676.875} C_VEL
LIN {X 0,Y 306.175,Z 543.662,A -85,B 0,C 180,E1 -16678.632,E2 -16678.632} C_VEL
LIN {X 0,Y 308.799,Z 529.989,A -85,B 0,C 180,E1 -16680.047,E2 -16680.047} C_VEL
LIN {X 0,Y 311.156,Z 515.829,A -85,B 0,C 180,E1 -16681.204,E2 -16681.204} C_VEL
LIN {X 0,Y 313.17,Z 501.25,A -85,B 0,C 180,E1 -16682.113,E2 -16682.113} C_VEL
LIN {X 0,Y 314.781,Z 486.282,A -85,B 0,C 180,E1 -16682.781,E2 -16682.781} C_VEL
LIN {X 0,Y 315.736,Z 470.867,A -85,B 0,C 180,E1 -16683.24,E2 -16683.24} C_VEL
LIN {X 0,Y 318.67,Z 392.078,A -85,B 0,C 180,E1 -16684.989,E2 -16684.989} C_VEL
LIN {X 0,Y 319.467,Z 368.813,A -85,B 0,C 180,E1 -16685.515,E2 -16685.515} C_VEL
LIN {X 0,Y 316.96,Z 353.852,A -85,B 0,C 180,E1 -16686.245,E2 -16686.245} C_VEL
LIN {X 0,Y 308.614,Z 335.359,A -85,B 0,C 180,E1 -16687.907,E2 -16687.907} C_VEL
LIN {X 0,Y 302.05,Z 322.575,A -85,B 0,C 180,E1 -16689.255,E2 -16689.255} C_VEL
LIN {X 0,Y 295.536,Z 310.458,A -85,B 0,C 180,E1 -16690.712,E2 -16690.712} C_VEL
LIN {X 0,Y 292.655,Z 301.064,A -85,B 0,C 180,E1 -16693.91,E2 -16693.91} C_VEL
LIN {X 0,Y 291.299,Z 296.814,A -85,B 0,C 180,E1 -16695.464,E2 -16695.464} C_VEL
LIN {X 0,Y 291.336,Z 296.817,A -85,B 0,C 180,E1 -16699.358,E2 -16699.358} C_VEL
LIN {X 0,Y 291.41,Z 296.808,A -85,B 0,C 180,E1 -16702.92,E2 -16702.92} C_VEL
LIN {X 0,Y 291.347,Z 296.816,A -85,B 0,C 180,E1 -16706.302,E2 -16706.302} C_VEL
LIN {X 0,Y 291.369,Z 296.806,A -85,B 0,C 180,E1 -16710.268,E2 -16710.268} C_VEL
LIN {X 0,Y 291.366,Z 296.807,A -85,B 0,C 180,E1 -16714.267,E2 -16714.267} C_VEL
LIN {X 0,Y 291.376,Z 296.804,A -85,B 0,C 180,E1 -16717.299,E2 -16717.299} C_VEL
LIN {X 0,Y 291.462,Z 296.797,A -85,B 0,C 180,E1 -16720.271,E2 -16720.271} C_VEL
LIN {X 0,Y 291.56,Z 296.783,A -85,B 0,C 180,E1 -16724.624,E2 -16724.624} C_VEL
LIN {X 0,Y 291.534,Z 296.785,A -85,B 0,C 180,E1 -16728.881,E2 -16728.881} C_VEL
LIN {X 0,Y 291.656,Z 296.777,A -85,B 0,C 180,E1 -16731.687,E2 -16731.687} C_VEL
LIN {X 0,Y 291.603,Z 296.787,A -85,B 0,C 180,E1 -16734.468,E2 -16734.468} C_VEL
LIN {X 0,Y 291.883,Z 296.751,A -85,B 0,C 180,E1 -16738.62,E2 -16738.62} C_VEL
LIN {X 0,Y 291.876,Z 296.744,A -85,B 0,C 180,E1 -16741.38,E2 -16741.38} C_VEL
LIN {X 0,Y 291.69,Z 296.769,A -85,B 0,C 180,E1 -16746.919,E2 -16746.919} C_VEL
LIN {X 0,Y 291.573,Z 296.783,A -85,B 0,C 180,E1 -16749.714,E2 -16749.714} C_VEL
LIN {X 0,Y 291.486,Z 296.794,A -85,B 0,C 180,E1 -16753.952,E2 -16753.952} C_VEL
LIN {X 0,Y 291.407,Z 296.811,A -85,B 0,C 180,E1 -16756.823,E2 -16756.823} C_VEL
LIN {X 0,Y 291.395,Z 296.809,A -85,B 0,C 180,E1 -16759.842,E2 -16759.842} C_VEL
LIN {X 0,Y 291.337,Z 296.82,A -85,B 0,C 180,E1 -16764.211,E2 -16764.211} C_VEL
LIN {X 0,Y 291.332,Z 296.792,A -85,B 0,C 180,E1 -16767.281,E2 -16767.281} C_VEL
LIN {X 0,Y 291.305,Z 296.819,A -85,B 0,C 180,E1 -16770.441,E2 -16770.441} C_VEL
LIN {X 0,Y 291.347,Z 296.815,A -85,B 0,C 180,E1 -16773.698,E2 -16773.698} C_VEL
LIN {X 0,Y 291.356,Z 296.817,A -85,B 0,C 180,E1 -16777.247,E2 -16777.247} C_VEL
LIN {X 0,Y 291.296,Z 296.822,A -85,B 0,C 180,E1 -16780.649,E2 -16780.649} C_VEL
LIN {X 0,Y 291.263,Z 296.825,A -85,B 0,C 180,E1 -16784.407,E2 -16784.407} C_VEL
LIN {X 0,Y 291.312,Z 296.914,A -85,B 0,C 180,E1 -16788.774,E2 -16788.774} C_VEL
LIN {X 0,Y 292.25,Z 299.57,A -85,B 0,C 180,E1 -16789.022,E2 -16789.022} C_VEL
LIN {X 0,Y 294.204,Z 302.075,A -85,B 0,C 180,E1 -16789.434,E2 -16789.434} C_VEL
LIN {X 0,Y 296.53,Z 305.553,A -85,B 0,C 180,E1 -16789.93,E2 -16789.93} C_VEL
LIN {X 0,Y 304.796,Z 318.633,A -85,B 0,C 180,E1 -16791.626,E2 -16791.626} C_VEL
LIN {X 0,Y 309.678,Z 327.155,A -85,B 0,C 180,E1 -16792.59,E2 -16792.59} C_VEL
LIN {X 0,Y 318.656,Z 345.643,A -85,B 0,C 180,E1 -16794.334,E2 -16794.334} C_VEL
LIN {X 0,Y 320.148,Z 349.108,A -85,B 0,C 180,E1 -16794.621,E2 -16794.621} C_VEL
LIN {X 0,Y 315.958,Z 458.233,A -85,B 0,C 180,E1 -16797.072,E2 -16797.072} C_VEL
LIN {X 0,Y 314.709,Z 474.177,A -85,B 0,C 180,E1 -16797.683,E2 -16797.683} C_VEL
LIN {X 0,Y 313.243,Z 488.57,A -85,B 0,C 180,E1 -16798.493,E2 -16798.493} C_VEL
LIN {X 0,Y 311.406,Z 501.987,A -85,B 0,C 180,E1 -16799.482,E2 -16799.482} C_VEL
LIN {X 0,Y 309.158,Z 515.535,A -85,B 0,C 180,E1 -16800.74,E2 -16800.74} C_VEL
LIN {X 0,Y 306.745,Z 527.996,A -85,B 0,C 180,E1 -16802.171,E2 -16802.171} C_VEL
LIN {X 0,Y 304.14,Z 539.557,A -85,B 0,C 180,E1 -16803.772,E2 -16803.772} C_VEL
LIN {X 0,Y 301.783,Z 550.28,A -85,B 0,C 180,E1 -16805.583,E2 -16805.583} C_VEL
LIN {X 0,Y 299.271,Z 560.197,A -85,B 0,C 180,E1 -16807.566,E2 -16807.566} C_VEL
LIN {X 0,Y 296.826,Z 569.872,A -85,B 0,C 180,E1 -16809.92,E2 -16809.92} C_VEL
LIN {X 0,Y 294.67,Z 578.117,A -85,B 0,C 180,E1 -16812.362,E2 -16812.362} C_VEL
LIN {X 0,Y 293.142,Z 584.573,A -85,B 0,C 180,E1 -16814.708,E2 -16814.708} C_VEL
LIN {X 0,Y 291.607,Z 590.722,A -85,B 0,C 180,E1 -16817.472,E2 -16817.472} C_VEL
LIN {X 0,Y 290.619,Z 595.462,A -85,B 0,C 180,E1 -16820.253,E2 -16820.253} C_VEL
LIN {X 0,Y 290.022,Z 598.929,A -85,B 0,C 180,E1 -16823.04,E2 -16823.04} C_VEL
LIN {X 0,Y 289.716,Z 601.218,A -85,B 0,C 180,E1 -16825.826,E2 -16825.826} C_VEL
LIN {X 0,Y 289.51,Z 602.388,A -85,B 0,C 180,E1 -16828.608,E2 -16828.608} C_VEL
LIN {X 0,Y 289.51,Z 602.402,A -85,B 0,C 180,E1 -16831.39,E2 -16831.39} C_VEL
LIN {X 0,Y 289.715,Z 601.287,A -85,B 0,C 180,E1 -16834.173,E2 -16834.173} C_VEL
LIN {X 0,Y 290.021,Z 599.051,A -85,B 0,C 180,E1 -16836.959,E2 -16836.959} C_VEL
LIN {X 0,Y 290.611,Z 595.633,A -85,B 0,C 180,E1 -16839.746,E2 -16839.746} C_VEL
LIN {X 0,Y 291.575,Z 590.95,A -85,B 0,C 180,E1 -16842.528,E2 -16842.528} C_VEL
LIN {X 0,Y 293.072,Z 584.871,A -85,B 0,C 180,E1 -16845.294,E2 -16845.294} C_VEL
LIN {X 0,Y 294.935,Z 577.215,A -85,B 0,C 180,E1 -16848.045,E2 -16848.045} C_VEL
LIN {X 0,Y 297.066,Z 569.042,A -85,B 0,C 180,E1 -16850.423,E2 -16850.423} C_VEL
LIN {X 0,Y 299.578,Z 559.191,A -85,B 0,C 180,E1 -16852.773,E2 -16852.773} C_VEL
LIN {X 0,Y 302.133,Z 548.469,A -85,B 0,C 180,E1 -16854.88,E2 -16854.88} C_VEL
LIN {X 0,Y 304.804,Z 537.045,A -85,B 0,C 180,E1 -16856.719,E2 -16856.719} C_VEL
LIN {X 0,Y 307.395,Z 524.962,A -85,B 0,C 180,E1 -16858.32,E2 -16858.32} C_VEL
LIN {X 0,Y 309.881,Z 511.825,A -85,B 0,C 180,E1 -16859.743,E2 -16859.743} C_VEL
LIN {X 0,Y 311.96,Z 498.255,A -85,B 0,C 180,E1 -16860.931,E2 -16860.931} C_VEL
LIN {X 0,Y 313.842,Z 483.343,A -85,B 0,C 180,E1 -16861.94,E2 -16861.94} C_VEL
LIN {X 0,Y 315.282,Z 468.45,A -85,B 0,C 180,E1 -16862.674,E2 -16862.674} C_VEL
LIN {X 0,Y 316.297,Z 453.11,A -85,B 0,C 180,E1 -16863.172,E2 -16863.172} C_VEL
LIN {X 0,Y 320.216,Z 349.239,A -85,B 0,C 180,E1 -16865.487,E2 -16865.487} C_VEL
LIN {X 0,Y 312.402,Z 332.386,A -85,B 0,C 180,E1 -16867,E2 -16867} C_VEL
LIN {X 0,Y 306.636,Z 321.599,A -85,B 0,C 180,E1 -16868.139,E2 -16868.139} C_VEL
LIN {X 0,Y 305.744,Z 320.112,A -85,B 0,C 180,E1 -16868.315,E2 -16868.315} C_VEL
LIN {X 0,Y 303.566,Z 317.603,A -85,B 0,C 180,E1 -16868.718,E2 -16868.718} C_VEL
LIN {X 0,Y 299.011,Z 314.971,A -85,B 0,C 180,E1 -16869.508,E2 -16869.508} C_VEL
LIN {X 0,Y 294.368,Z 312.515,A -85,B 0,C 180,E1 -16870.342,E2 -16870.342} C_VEL
LIN {X 0,Y 292.043,Z 310.249,A -85,B 0,C 180,E1 -16870.806,E2 -16870.806} C_VEL
LIN {X 0,Y 288.512,Z 305.181,A -85,B 0,C 180,E1 -16871.585,E2 -16871.585} C_VEL
LIN {X 0,Y 286.751,Z 302.283,A -85,B 0,C 180,E1 -16871.997,E2 -16871.997} C_VEL
LIN {X 0,Y 284.98,Z 300.026,A -85,B 0,C 180,E1 -16872.396,E2 -16872.396} C_VEL
LIN {X 0,Y 284.259,Z 297.684,A -85,B 0,C 180,E1 -16872.637,E2 -16872.637} C_VEL
LIN {X 0,Y 284.235,Z 297.695,A -85,B 0,C 180,E1 -16876.185,E2 -16876.185} C_VEL
LIN {X 0,Y 284.254,Z 297.7,A -85,B 0,C 180,E1 -16880.036,E2 -16880.036} C_VEL
LIN {X 0,Y 284.316,Z 297.661,A -85,B 0,C 180,E1 -16883.611,E2 -16883.611} C_VEL
LIN {X 0,Y 284.303,Z 297.696,A -85,B 0,C 180,E1 -16887.19,E2 -16887.19} C_VEL
LIN {X 0,Y 284.306,Z 297.696,A -85,B 0,C 180,E1 -16890.37,E2 -16890.37} C_VEL
LIN {X 0,Y 284.293,Z 297.693,A -85,B 0,C 180,E1 -16893.578,E2 -16893.578} C_VEL
LIN {X 0,Y 284.306,Z 297.685,A -85,B 0,C 180,E1 -16896.702,E2 -16896.702} C_VEL
LIN {X 0,Y 284.332,Z 297.688,A -85,B 0,C 180,E1 -16899.928,E2 -16899.928} C_VEL
LIN {X 0,Y 284.412,Z 297.678,A -85,B 0,C 180,E1 -16904.516,E2 -16904.516} C_VEL
LIN {X 0,Y 284.477,Z 297.675,A -85,B 0,C 180,E1 -16908.601,E2 -16908.601} C_VEL
LIN {X 0,Y 284.606,Z 297.646,A -85,B 0,C 180,E1 -16911.479,E2 -16911.479} C_VEL
LIN {X 0,Y 284.568,Z 297.659,A -85,B 0,C 180,E1 -16914.33,E2 -16914.33} C_VEL
LIN {X 0,Y 284.84,Z 297.63,A -85,B 0,C 180,E1 -16918.586,E2 -16918.586} C_VEL
LIN {X 0,Y 284.844,Z 297.614,A -85,B 0,C 180,E1 -16921.414,E2 -16921.414} C_VEL
LIN {X 0,Y 284.641,Z 297.647,A -85,B 0,C 180,E1 -16927.091,E2 -16927.091} C_VEL
LIN {X 0,Y 284.512,Z 297.661,A -85,B 0,C 180,E1 -16929.957,E2 -16929.957} C_VEL
LIN {X 0,Y 284.48,Z 297.667,A -85,B 0,C 180,E1 -16934.303,E2 -16934.303} C_VEL
LIN {X 0,Y 284.424,Z 297.682,A -85,B 0,C 180,E1 -16937.248,E2 -16937.248} C_VEL
LIN {X 0,Y 284.378,Z 297.681,A -85,B 0,C 180,E1 -16940.242,E2 -16940.242} C_VEL
LIN {X 0,Y 284.322,Z 297.667,A -85,B 0,C 180,E1 -16943.855,E2 -16943.855} C_VEL
LIN {X 0,Y 284.286,Z 297.694,A -85,B 0,C 180,E1 -16948.015,E2 -16948.015} C_VEL
LIN {X 0,Y 284.283,Z 297.67,A -85,B 0,C 180,E1 -16951.276,E2 -16951.276} C_VEL
LIN {X 0,Y 284.339,Z 297.689,A -85,B 0,C 180,E1 -16955.348,E2 -16955.348} C_VEL
LIN {X 0,Y 284.306,Z 297.674,A -85,B 0,C 180,E1 -16958.17,E2 -16958.17} C_VEL
LIN {X 0,Y 284.267,Z 297.702,A -85,B 0,C 180,E1 -16962.125,E2 -16962.125} C_VEL
LIN {X 0,Y 284.278,Z 297.731,A -85,B 0,C 180,E1 -16963.465,E2 -16963.465} C_VEL
LIN {X 0,Y 287.462,Z 307.817,A -85,B 0,C 180,E1 -16967.176,E2 -16967.176} C_VEL
LIN {X 0,Y 288.239,Z 310.342,A -85,B 0,C 180,E1 -16968.045,E2 -16968.045} C_VEL
LIN {X 0,Y 296.638,Z 325.42,A -85,B 0,C 180,E1 -16969.942,E2 -16969.942} C_VEL
LIN {X 0,Y 304.292,Z 340.49,A -85,B 0,C 180,E1 -16971.577,E2 -16971.577} C_VEL
LIN {X 0,Y 311.848,Z 357.72,A -85,B 0,C 180,E1 -16973.147,E2 -16973.147} C_VEL
LIN {X 0,Y 313.737,Z 370.178,A -85,B 0,C 180,E1 -16973.749,E2 -16973.749} C_VEL
LIN {X 0,Y 310.354,Z 459.266,A -85,B 0,C 180,E1 -16975.766,E2 -16975.766} C_VEL
LIN {X 0,Y 309.249,Z 481.11,A -85,B 0,C 180,E1 -16976.314,E2 -16976.314} C_VEL
LIN {X 0,Y 307.748,Z 496.895,A -85,B 0,C 180,E1 -16976.96,E2 -16976.96} C_VEL
LIN {X 0,Y 305.759,Z 511.392,A -85,B 0,C 180,E1 -16977.794,E2 -16977.794} C_VEL
LIN {X 0,Y 303.507,Z 525.385,A -85,B 0,C 180,E1 -16978.87,E2 -16978.87} C_VEL
LIN {X 0,Y 301.09,Z 538.177,A -85,B 0,C 180,E1 -16980.11,E2 -16980.11} C_VEL
LIN {X 0,Y 298.211,Z 551.332,A -85,B 0,C 180,E1 -16981.687,E2 -16981.687} C_VEL
LIN {X 0,Y 295.292,Z 563.584,A -85,B 0,C 180,E1 -16983.497,E2 -16983.497} C_VEL
LIN {X 0,Y 292.498,Z 574.782,A -85,B 0,C 180,E1 -16985.514,E2 -16985.514} C_VEL
LIN {X 0,Y 289.776,Z 585.658,A -85,B 0,C 180,E1 -16987.919,E2 -16987.919} C_VEL
LIN {X 0,Y 287.45,Z 594.724,A -85,B 0,C 180,E1 -16990.356,E2 -16990.356} C_VEL
LIN {X 0,Y 285.562,Z 602.251,A -85,B 0,C 180,E1 -16992.823,E2 -16992.823} C_VEL
LIN {X 0,Y 284.066,Z 609.286,A -85,B 0,C 180,E1 -16995.677,E2 -16995.677} C_VEL
LIN {X 0,Y 283.029,Z 614.824,A -85,B 0,C 180,E1 -16998.543,E2 -16998.543} C_VEL
LIN {X 0,Y 282.532,Z 619.021,A -85,B 0,C 180,E1 -17001.417,E2 -17001.417} C_VEL
LIN {X 0,Y 282.381,Z 621.97,A -85,B 0,C 180,E1 -17004.287,E2 -17004.287} C_VEL
LIN {X 0,Y 282.373,Z 623.73,A -85,B 0,C 180,E1 -17007.147,E2 -17007.147} C_VEL
LIN {X 0,Y 282.411,Z 624.332,A -85,B 0,C 180,E1 -17010.001,E2 -17010.001} C_VEL
LIN {X 0,Y 282.373,Z 623.719,A -85,B 0,C 180,E1 -17012.854,E2 -17012.854} C_VEL
LIN {X 0,Y 282.374,Z 621.945,A -85,B 0,C 180,E1 -17015.714,E2 -17015.714} C_VEL
LIN {X 0,Y 282.531,Z 618.987,A -85,B 0,C 180,E1 -17018.584,E2 -17018.584} C_VEL
LIN {X 0,Y 283.022,Z 614.782,A -85,B 0,C 180,E1 -17021.459,E2 -17021.459} C_VEL
LIN {X 0,Y 284.068,Z 609.227,A -85,B 0,C 180,E1 -17024.325,E2 -17024.325} C_VEL
LIN {X 0,Y 285.562,Z 602.169,A -85,B 0,C 180,E1 -17027.178,E2 -17027.178} C_VEL
LIN {X 0,Y 287.367,Z 594.629,A -85,B 0,C 180,E1 -17029.651,E2 -17029.651} C_VEL
LIN {X 0,Y 289.788,Z 585.555,A -85,B 0,C 180,E1 -17032.081,E2 -17032.081} C_VEL
LIN {X 0,Y 292.054,Z 576.294,A -85,B 0,C 180,E1 -17034.148,E2 -17034.148} C_VEL
LIN {X 0,Y 294.755,Z 565.395,A -85,B 0,C 180,E1 -17036.175,E2 -17036.175} C_VEL
LIN {X 0,Y 297.606,Z 553.51,A -85,B 0,C 180,E1 -17037.993,E2 -17037.993} C_VEL
LIN {X 0,Y 300.539,Z 540.628,A -85,B 0,C 180,E1 -17039.591,E2 -17039.591} C_VEL
LIN {X 0,Y 303.241,Z 526.528,A -85,B 0,C 180,E1 -17041.004,E2 -17041.004} C_VEL
LIN {X 0,Y 305.556,Z 512.159,A -85,B 0,C 180,E1 -17042.134,E2 -17042.134} C_VEL
LIN {X 0,Y 307.62,Z 497.173,A -85,B 0,C 180,E1 -17043.008,E2 -17043.008} C_VEL
LIN {X 0,Y 309.159,Z 481.505,A -85,B 0,C 180,E1 -17043.65,E2 -17043.65} C_VEL
LIN {X 0,Y 310.154,Z 461.656,A -85,B 0,C 180,E1 -17044.163,E2 -17044.163} C_VEL
LIN {X 0,Y 312.922,Z 390.031,A -85,B 0,C 180,E1 -17045.778,E2 -17045.778} C_VEL
LIN {X 0,Y 313.669,Z 369.962,A -85,B 0,C 180,E1 -17046.234,E2 -17046.234} C_VEL
LIN {X 0,Y 311.419,Z 356.703,A -85,B 0,C 180,E1 -17046.907,E2 -17046.907} C_VEL
LIN {X 0,Y 303.803,Z 339.564,A -85,B 0,C 180,E1 -17048.486,E2 -17048.486} C_VEL
LIN {X 0,Y 297.762,Z 327.62,A -85,B 0,C 180,E1 -17049.771,E2 -17049.771} C_VEL
LIN {X 0,Y 290.627,Z 314.634,A -85,B 0,C 180,E1 -17051.355,E2 -17051.355} C_VEL
LIN {X 0,Y 288.207,Z 310.281,A -85,B 0,C 180,E1 -17051.923,E2 -17051.923} C_VEL
LIN {X 0,Y 284.907,Z 299.882,A -85,B 0,C 180,E1 -17055.674,E2 -17055.674} C_VEL
LIN {X 0,Y 284.261,Z 297.684,A -85,B 0,C 180,E1 -17056.532,E2 -17056.532} C_VEL
LIN {X 0,Y 284.31,Z 297.691,A -85,B 0,C 180,E1 -17060.025,E2 -17060.025} C_VEL
LIN {X 0,Y 284.336,Z 297.691,A -85,B 0,C 180,E1 -17063.615,E2 -17063.615} C_VEL
LIN {X 0,Y 284.309,Z 297.686,A -85,B 0,C 180,E1 -17067.191,E2 -17067.191} C_VEL
LIN {X 0,Y 284.341,Z 297.681,A -85,B 0,C 180,E1 -17070.374,E2 -17070.374} C_VEL
LIN {X 0,Y 284.31,Z 297.685,A -85,B 0,C 180,E1 -17073.58,E2 -17073.58} C_VEL
LIN {X 0,Y 284.334,Z 297.683,A -85,B 0,C 180,E1 -17076.704,E2 -17076.704} C_VEL
LIN {X 0,Y 284.403,Z 297.674,A -85,B 0,C 180,E1 -17081.262,E2 -17081.262} C_VEL
LIN {X 0,Y 284.497,Z 297.663,A -85,B 0,C 180,E1 -17084.46,E2 -17084.46} C_VEL
LIN {X 0,Y 284.488,Z 297.663,A -85,B 0,C 180,E1 -17088.602,E2 -17088.602} C_VEL
LIN {X 0,Y 284.613,Z 297.657,A -85,B 0,C 180,E1 -17091.48,E2 -17091.48} C_VEL
LIN {X 0,Y 284.573,Z 297.661,A -85,B 0,C 180,E1 -17094.331,E2 -17094.331} C_VEL
LIN {X 0,Y 284.849,Z 297.626,A -85,B 0,C 180,E1 -17098.586,E2 -17098.586} C_VEL
LIN {X 0,Y 284.844,Z 297.62,A -85,B 0,C 180,E1 -17101.414,E2 -17101.414} C_VEL
LIN {X 0,Y 284.646,Z 297.647,A -85,B 0,C 180,E1 -17107.092,E2 -17107.092} C_VEL
LIN {X 0,Y 284.518,Z 297.66,A -85,B 0,C 180,E1 -17109.957,E2 -17109.957} C_VEL
LIN {X 0,Y 284.423,Z 297.671,A -85,B 0,C 180,E1 -17114.306,E2 -17114.306} C_VEL
LIN {X 0,Y 284.321,Z 297.684,A -85,B 0,C 180,E1 -17118.744,E2 -17118.744} C_VEL
LIN {X 0,Y 284.301,Z 297.692,A -85,B 0,C 180,E1 -17121.765,E2 -17121.765} C_VEL
LIN {X 0,Y 284.292,Z 297.698,A -85,B 0,C 180,E1 -17124.851,E2 -17124.851} C_VEL
LIN {X 0,Y 284.263,Z 297.669,A -85,B 0,C 180,E1 -17128.018,E2 -17128.018} C_VEL
LIN {X 0,Y 284.282,Z 297.7,A -85,B 0,C 180,E1 -17131.276,E2 -17131.276} C_VEL
LIN {X 0,Y 284.34,Z 297.687,A -85,B 0,C 180,E1 -17135.346,E2 -17135.346} C_VEL
LIN {X 0,Y 284.298,Z 297.692,A -85,B 0,C 180,E1 -17138.171,E2 -17138.171} C_VEL
LIN {X 0,Y 284.233,Z 297.701,A -85,B 0,C 180,E1 -17142.115,E2 -17142.115} C_VEL
LIN {X 0,Y 284.21,Z 297.703,A -85,B 0,C 180,E1 -17146.179,E2 -17146.179} C_VEL
LIN {X 0,Y 284.253,Z 297.818,A -85,B 0,C 180,E1 -17147.533,E2 -17147.533} C_VEL
LIN {X 0,Y 285.266,Z 300.614,A -85,B 0,C 180,E1 -17147.814,E2 -17147.814} C_VEL
LIN {X 0,Y 287.26,Z 303.009,A -85,B 0,C 180,E1 -17148.256,E2 -17148.256} C_VEL
LIN {X 0,Y 289.466,Z 306.394,A -85,B 0,C 180,E1 -17148.759,E2 -17148.759} C_VEL
LIN {X 0,Y 299.275,Z 321.505,A -85,B 0,C 180,E1 -17150.863,E2 -17150.863} C_VEL
LIN {X 0,Y 304.821,Z 331.295,A -85,B 0,C 180,E1 -17152.003,E2 -17152.003} C_VEL
LIN {X 0,Y 313.484,Z 349.275,A -85,B 0,C 180,E1 -17153.746,E2 -17153.746} C_VEL
LIN {X 0,Y 314.31,Z 351.261,A -85,B 0,C 180,E1 -17153.913,E2 -17153.913} C_VEL
LIN {X 0,Y 310.109,Z 457.099,A -85,B 0,C 180,E1 -17156.32,E2 -17156.32} C_VEL
LIN {X 0,Y 309.003,Z 471.904,A -85,B 0,C 180,E1 -17156.867,E2 -17156.867} C_VEL
LIN {X 0,Y 307.562,Z 485.604,A -85,B 0,C 180,E1 -17157.598,E2 -17157.598} C_VEL
LIN {X 0,Y 305.607,Z 500.286,A -85,B 0,C 180,E1 -17158.646,E2 -17158.646} C_VEL
LIN {X 0,Y 303.272,Z 514.235,A -85,B 0,C 180,E1 -17159.924,E2 -17159.924} C_VEL
LIN {X 0,Y 300.765,Z 526.985,A -85,B 0,C 180,E1 -17161.377,E2 -17161.377} C_VEL
LIN {X 0,Y 297.788,Z 539.831,A -85,B 0,C 180,E1 -17163.168,E2 -17163.168} C_VEL
LIN {X 0,Y 295.285,Z 550.624,A -85,B 0,C 180,E1 -17165.024,E2 -17165.024} C_VEL
LIN {X 0,Y 292.71,Z 560.47,A -85,B 0,C 180,E1 -17167.034,E2 -17167.034} C_VEL
LIN {X 0,Y 290.129,Z 570.146,A -85,B 0,C 180,E1 -17169.436,E2 -17169.436} C_VEL
LIN {X 0,Y 287.822,Z 578.567,A -85,B 0,C 180,E1 -17171.993,E2 -17171.993} C_VEL
LIN {X 0,Y 286.273,Z 584.846,A -85,B 0,C 180,E1 -17174.332,E2 -17174.332} C_VEL
LIN {X 0,Y 284.639,Z 590.995,A -85,B 0,C 180,E1 -17177.16,E2 -17177.16} C_VEL
LIN {X 0,Y 283.612,Z 595.734,A -85,B 0,C 180,E1 -17180.01,E2 -17180.01} C_VEL
LIN {X 0,Y 282.973,Z 599.2,A -85,B 0,C 180,E1 -17182.866,E2 -17182.866} C_VEL
LIN {X 0,Y 282.635,Z 601.489,A -85,B 0,C 180,E1 -17185.721,E2 -17185.721} C_VEL
LIN {X 0,Y 282.431,Z 602.658,A -85,B 0,C 180,E1 -17188.573,E2 -17188.573} C_VEL
LIN {X 0,Y 282.431,Z 602.671,A -85,B 0,C 180,E1 -17191.425,E2 -17191.425} C_VEL
LIN {X 0,Y 282.634,Z 601.557,A -85,B 0,C 180,E1 -17194.277,E2 -17194.277} C_VEL
LIN {X 0,Y 282.972,Z 599.321,A -85,B 0,C 180,E1 -17197.133,E2 -17197.133} C_VEL
LIN {X 0,Y 283.603,Z 595.904,A -85,B 0,C 180,E1 -17199.989,E2 -17199.989} C_VEL
LIN {X 0,Y 284.607,Z 591.221,A -85,B 0,C 180,E1 -17202.84,E2 -17202.84} C_VEL
LIN {X 0,Y 286.204,Z 585.141,A -85,B 0,C 180,E1 -17205.67,E2 -17205.67} C_VEL
LIN {X 0,Y 288.162,Z 577.485,A -85,B 0,C 180,E1 -17208.484,E2 -17208.484} C_VEL
LIN {X 0,Y 290.384,Z 569.312,A -85,B 0,C 180,E1 -17210.915,E2 -17210.915} C_VEL
LIN {X 0,Y 293.035,Z 559.459,A -85,B 0,C 180,E1 -17213.311,E2 -17213.311} C_VEL
LIN {X 0,Y 295.586,Z 549.177,A -85,B 0,C 180,E1 -17215.377,E2 -17215.377} C_VEL
LIN {X 0,Y 298.488,Z 537.312,A -85,B 0,C 180,E1 -17217.331,E2 -17217.331} C_VEL
LIN {X 0,Y 301.148,Z 525.229,A -85,B 0,C 180,E1 -17218.963,E2 -17218.963} C_VEL
LIN {X 0,Y 303.719,Z 512.091,A -85,B 0,C 180,E1 -17220.409,E2 -17220.409} C_VEL
LIN {X 0,Y 305.818,Z 499.036,A -85,B 0,C 180,E1 -17221.572,E2 -17221.572} C_VEL
LIN {X 0,Y 307.759,Z 484.374,A -85,B 0,C 180,E1 -17222.591,E2 -17222.591} C_VEL
LIN {X 0,Y 309.261,Z 469.621,A -85,B 0,C 180,E1 -17223.343,E2 -17223.343} C_VEL
LIN {X 0,Y 310.289,Z 454.863,A -85,B 0,C 180,E1 -17223.851,E2 -17223.851} C_VEL
LIN {X 0,Y 314.406,Z 352.666,A -85,B 0,C 180,E1 -17226.157,E2 -17226.157} C_VEL
LIN {X 0,Y 314.16,Z 350.901,A -85,B 0,C 180,E1 -17226.24,E2 -17226.24} C_VEL
LIN {X 0,Y 306.499,Z 334.484,A -85,B 0,C 180,E1 -17227.783,E2 -17227.783} C_VEL
LIN {X 0,Y 301.911,Z 325.96,A -85,B 0,C 180,E1 -17228.722,E2 -17228.722} C_VEL
LIN {X 0,Y 294.198,Z 313.551,A -85,B 0,C 180,E1 -17230.337,E2 -17230.337} C_VEL
LIN {X 0,Y 292.043,Z 310.249,A -85,B 0,C 180,E1 -17230.806,E2 -17230.806} C_VEL
LIN {X 0,Y 289.706,Z 308.076,A -85,B 0,C 180,E1 -17231.28,E2 -17231.28} C_VEL
LIN {X 0,Y 280.551,Z 303.929,A -85,B 0,C 180,E1 -17233.1,E2 -17233.1} C_VEL
LIN {X 0,Y 278.384,Z 301.672,A -85,B 0,C 180,E1 -17233.602,E2 -17233.602} C_VEL
LIN {X 0,Y 277.33,Z 299.311,A -85,B 0,C 180,E1 -17233.895,E2 -17233.895} C_VEL
LIN {X 0,Y 277.198,Z 298.565,A -85,B 0,C 180,E1 -17233.958,E2 -17233.958} C_VEL
LIN {X 0,Y 277.19,Z 298.558,A -85,B 0,C 180,E1 -17237.33,E2 -17237.33} C_VEL
LIN {X 0,Y 277.221,Z 298.563,A -85,B 0,C 180,E1 -17241.803,E2 -17241.803} C_VEL
LIN {X 0,Y 277.274,Z 298.539,A -85,B 0,C 180,E1 -17244.34,E2 -17244.34} C_VEL
LIN {X 0,Y 277.234,Z 298.573,A -85,B 0,C 180,E1 -17247.835,E2 -17247.835} C_VEL
LIN {X 0,Y 277.214,Z 298.578,A -85,B 0,C 180,E1 -17251.204,E2 -17251.204} C_VEL
LIN {X 0,Y 277.23,Z 298.578,A -85,B 0,C 180,E1 -17254.471,E2 -17254.471} C_VEL
LIN {X 0,Y 277.245,Z 298.568,A -85,B 0,C 180,E1 -17257.651,E2 -17257.651} C_VEL
LIN {X 0,Y 277.274,Z 298.559,A -85,B 0,C 180,E1 -17260.761,E2 -17260.761} C_VEL
LIN {X 0,Y 277.369,Z 298.548,A -85,B 0,C 180,E1 -17265.322,E2 -17265.322} C_VEL
LIN {X 0,Y 277.455,Z 298.541,A -85,B 0,C 180,E1 -17269.787,E2 -17269.787} C_VEL
LIN {X 0,Y 277.598,Z 298.53,A -85,B 0,C 180,E1 -17272.727,E2 -17272.727} C_VEL
LIN {X 0,Y 277.807,Z 298.506,A -85,B 0,C 180,E1 -17278.55,E2 -17278.55} C_VEL
LIN {X 0,Y 277.81,Z 298.49,A -85,B 0,C 180,E1 -17281.449,E2 -17281.449} C_VEL
LIN {X 0,Y 277.599,Z 298.526,A -85,B 0,C 180,E1 -17287.272,E2 -17287.272} C_VEL
LIN {X 0,Y 277.456,Z 298.538,A -85,B 0,C 180,E1 -17290.213,E2 -17290.213} C_VEL
LIN {X 0,Y 277.433,Z 298.542,A -85,B 0,C 180,E1 -17294.674,E2 -17294.674} C_VEL
LIN {X 0,Y 277.343,Z 298.555,A -85,B 0,C 180,E1 -17299.234,E2 -17299.234} C_VEL
LIN {X 0,Y 277.275,Z 298.569,A -85,B 0,C 180,E1 -17302.346,E2 -17302.346} C_VEL
LIN {X 0,Y 277.251,Z 298.536,A -85,B 0,C 180,E1 -17305.527,E2 -17305.527} C_VEL
LIN {X 0,Y 277.241,Z 298.576,A -85,B 0,C 180,E1 -17308.793,E2 -17308.793} C_VEL
LIN {X 0,Y 277.238,Z 298.545,A -85,B 0,C 180,E1 -17312.164,E2 -17312.164} C_VEL
LIN {X 0,Y 277.278,Z 298.562,A -85,B 0,C 180,E1 -17315.799,E2 -17315.799} C_VEL
LIN {X 0,Y 277.231,Z 298.57,A -85,B 0,C 180,E1 -17319.328,E2 -17319.328} C_VEL
LIN {X 0,Y 277.244,Z 298.652,A -85,B 0,C 180,E1 -17322.346,E2 -17322.346} C_VEL
LIN {X 0,Y 280.905,Z 310.11,A -85,B 0,C 180,E1 -17326.689,E2 -17326.689} C_VEL
LIN {X 0,Y 283.706,Z 314.847,A -85,B 0,C 180,E1 -17327.375,E2 -17327.375} C_VEL
LIN {X 0,Y 291.973,Z 329.631,A -85,B 0,C 180,E1 -17329.308,E2 -17329.308} C_VEL
LIN {X 0,Y 299.146,Z 343.927,A -85,B 0,C 180,E1 -17330.902,E2 -17330.902} C_VEL
LIN {X 0,Y 306.377,Z 360.394,A -85,B 0,C 180,E1 -17332.46,E2 -17332.46} C_VEL
LIN {X 0,Y 307.996,Z 371.304,A -85,B 0,C 180,E1 -17333.001,E2 -17333.001} C_VEL
LIN {X 0,Y 304.419,Z 460.807,A -85,B 0,C 180,E1 -17335.052,E2 -17335.052} C_VEL
LIN {X 0,Y 303.368,Z 480.853,A -85,B 0,C 180,E1 -17335.57,E2 -17335.57} C_VEL
LIN {X 0,Y 301.829,Z 496.634,A -85,B 0,C 180,E1 -17336.226,E2 -17336.226} C_VEL
LIN {X 0,Y 299.771,Z 511.128,A -85,B 0,C 180,E1 -17337.07,E2 -17337.07} C_VEL
LIN {X 0,Y 297.559,Z 524.435,A -85,B 0,C 180,E1 -17338.099,E2 -17338.099} C_VEL
LIN {X 0,Y 295.139,Z 536.981,A -85,B 0,C 180,E1 -17339.316,E2 -17339.316} C_VEL
LIN {X 0,Y 292.243,Z 549.852,A -85,B 0,C 180,E1 -17340.858,E2 -17340.858} C_VEL
LIN {X 0,Y 289.186,Z 562.299,A -85,B 0,C 180,E1 -17342.697,E2 -17342.697} C_VEL
LIN {X 0,Y 285.966,Z 574.51,A -85,B 0,C 180,E1 -17344.917,E2 -17344.917} C_VEL
LIN {X 0,Y 283.467,Z 583.942,A -85,B 0,C 180,E1 -17347.016,E2 -17347.016} C_VEL
LIN {X 0,Y 280.962,Z 593.227,A -85,B 0,C 180,E1 -17349.501,E2 -17349.501} C_VEL
LIN {X 0,Y 278.714,Z 601.979,A -85,B 0,C 180,E1 -17352.387,E2 -17352.387} C_VEL
LIN {X 0,Y 277.122,Z 609.014,A -85,B 0,C 180,E1 -17355.31,E2 -17355.31} C_VEL
LIN {X 0,Y 276.012,Z 614.552,A -85,B 0,C 180,E1 -17358.247,E2 -17358.247} C_VEL
LIN {X 0,Y 275.454,Z 618.749,A -85,B 0,C 180,E1 -17361.195,E2 -17361.195} C_VEL
LIN {X 0,Y 275.292,Z 621.699,A -85,B 0,C 180,E1 -17364.14,E2 -17364.14} C_VEL
LIN {X 0,Y 275.279,Z 623.459,A -85,B 0,C 180,E1 -17367.074,E2 -17367.074} C_VEL
LIN {X 0,Y 275.33,Z 624.062,A -85,B 0,C 180,E1 -17370.001,E2 -17370.001} C_VEL
LIN {X 0,Y 275.279,Z 623.448,A -85,B 0,C 180,E1 -17372.928,E2 -17372.928} C_VEL
LIN {X 0,Y 275.287,Z 621.673,A -85,B 0,C 180,E1 -17375.862,E2 -17375.862} C_VEL
LIN {X 0,Y 275.453,Z 618.713,A -85,B 0,C 180,E1 -17378.807,E2 -17378.807} C_VEL
LIN {X 0,Y 276.006,Z 614.508,A -85,B 0,C 180,E1 -17381.754,E2 -17381.754} C_VEL
LIN {X 0,Y 277.124,Z 608.953,A -85,B 0,C 180,E1 -17384.692,E2 -17384.692} C_VEL
LIN {X 0,Y 278.715,Z 601.894,A -85,B 0,C 180,E1 -17387.614,E2 -17387.614} C_VEL
LIN {X 0,Y 280.927,Z 593.125,A -85,B 0,C 180,E1 -17390.503,E2 -17390.503} C_VEL
LIN {X 0,Y 283.478,Z 583.824,A -85,B 0,C 180,E1 -17392.985,E2 -17392.985} C_VEL
LIN {X 0,Y 285.981,Z 574.375,A -85,B 0,C 180,E1 -17395.083,E2 -17395.083} C_VEL
LIN {X 0,Y 289.122,Z 562.126,A -85,B 0,C 180,E1 -17397.312,E2 -17397.312} C_VEL
LIN {X 0,Y 292.178,Z 549.646,A -85,B 0,C 180,E1 -17399.15,E2 -17399.15} C_VEL
LIN {X 0,Y 295.117,Z 536.772,A -85,B 0,C 180,E1 -17400.682,E2 -17400.682} C_VEL
LIN {X 0,Y 297.854,Z 522.293,A -85,B 0,C 180,E1 -17402.066,E2 -17402.066} C_VEL
LIN {X 0,Y 300.26,Z 507.224,A -85,B 0,C 180,E1 -17403.171,E2 -17403.171} C_VEL
LIN {X 0,Y 302.273,Z 492.147,A -85,B 0,C 180,E1 -17403.97,E2 -17403.97} C_VEL
LIN {X 0,Y 303.626,Z 476.322,A -85,B 0,C 180,E1 -17404.549,E2 -17404.549} C_VEL
LIN {X 0,Y 306.675,Z 402.867,A -85,B 0,C 180,E1 -17406.25,E2 -17406.25} C_VEL
LIN {X 0,Y 307.922,Z 371.119,A -85,B 0,C 180,E1 -17406.981,E2 -17406.981} C_VEL
LIN {X 0,Y 306.079,Z 359.854,A -85,B 0,C 180,E1 -17407.563,E2 -17407.563} C_VEL
LIN {X 0,Y 297.752,Z 340.998,A -85,B 0,C 180,E1 -17409.364,E2 -17409.364} C_VEL
LIN {X 0,Y 288.819,Z 323.861,A -85,B 0,C 180,E1 -17411.369,E2 -17411.369} C_VEL
LIN {X 0,Y 282.927,Z 313.754,A -85,B 0,C 180,E1 -17412.758,E2 -17412.758} C_VEL
LIN {X 0,Y 280.823,Z 309.878,A -85,B 0,C 180,E1 -17413.297,E2 -17413.297} C_VEL
LIN {X 0,Y 277.226,Z 298.566,A -85,B 0,C 180,E1 -17417.654,E2 -17417.654} C_VEL
LIN {X 0,Y 277.268,Z 298.567,A -85,B 0,C 180,E1 -17421.793,E2 -17421.793} C_VEL
LIN {X 0,Y 277.288,Z 298.563,A -85,B 0,C 180,E1 -17424.342,E2 -17424.342} C_VEL
LIN {X 0,Y 277.243,Z 298.565,A -85,B 0,C 180,E1 -17427.836,E2 -17427.836} C_VEL
LIN {X 0,Y 277.243,Z 298.566,A -85,B 0,C 180,E1 -17431.207,E2 -17431.207} C_VEL
LIN {X 0,Y 277.252,Z 298.566,A -85,B 0,C 180,E1 -17434.474,E2 -17434.474} C_VEL
LIN {X 0,Y 277.271,Z 298.562,A -85,B 0,C 180,E1 -17437.654,E2 -17437.654} C_VEL
LIN {X 0,Y 277.347,Z 298.553,A -85,B 0,C 180,E1 -17440.766,E2 -17440.766} C_VEL
LIN {X 0,Y 277.44,Z 298.543,A -85,B 0,C 180,E1 -17445.326,E2 -17445.326} C_VEL
LIN {X 0,Y 277.462,Z 298.542,A -85,B 0,C 180,E1 -17449.787,E2 -17449.787} C_VEL
LIN {X 0,Y 277.605,Z 298.519,A -85,B 0,C 180,E1 -17452.728,E2 -17452.728} C_VEL
LIN {X 0,Y 277.815,Z 298.502,A -85,B 0,C 180,E1 -17458.551,E2 -17458.551} C_VEL
LIN {X 0,Y 277.811,Z 298.495,A -85,B 0,C 180,E1 -17461.45,E2 -17461.45} C_VEL
LIN {X 0,Y 277.604,Z 298.525,A -85,B 0,C 180,E1 -17467.272,E2 -17467.272} C_VEL
LIN {X 0,Y 277.459,Z 298.538,A -85,B 0,C 180,E1 -17470.213,E2 -17470.213} C_VEL
LIN {X 0,Y 277.375,Z 298.548,A -85,B 0,C 180,E1 -17474.677,E2 -17474.677} C_VEL
LIN {X 0,Y 277.28,Z 298.562,A -85,B 0,C 180,E1 -17479.239,E2 -17479.239} C_VEL
LIN {X 0,Y 277.264,Z 298.571,A -85,B 0,C 180,E1 -17483.927,E2 -17483.927} C_VEL
LIN {X 0,Y 277.239,Z 298.545,A -85,B 0,C 180,E1 -17487.468,E2 -17487.468} C_VEL
LIN {X 0,Y 277.232,Z 298.571,A -85,B 0,C 180,E1 -17490.465,E2 -17490.465} C_VEL
LIN {X 0,Y 277.249,Z 298.573,A -85,B 0,C 180,E1 -17493.896,E2 -17493.896} C_VEL
LIN {X 0,Y 277.254,Z 298.574,A -85,B 0,C 180,E1 -17497.472,E2 -17497.472} C_VEL
LIN {X 0,Y 277.182,Z 298.576,A -85,B 0,C 180,E1 -17501.242,E2 -17501.242} C_VEL
LIN {X 0,Y 277.157,Z 298.585,A -85,B 0,C 180,E1 -17505.236,E2 -17505.236} C_VEL
LIN {X 0,Y 277.166,Z 298.58,A -85,B 0,C 180,E1 -17506.176,E2 -17506.176} C_VEL
LIN {X 0,Y 278.189,Z 301.443,A -85,B 0,C 180,E1 -17506.494,E2 -17506.494} C_VEL
LIN {X 0,Y 280.255,Z 303.886,A -85,B 0,C 180,E1 -17506.982,E2 -17506.982} C_VEL
LIN {X 0,Y 282.389,Z 307.224,A -85,B 0,C 180,E1 -17507.502,E2 -17507.502} C_VEL
LIN {X 0,Y 289.231,Z 317.471,A -85,B 0,C 180,E1 -17509.076,E2 -17509.076} C_VEL
LIN {X 0,Y 295.452,Z 327.333,A -85,B 0,C 180,E1 -17510.431,E2 -17510.431} C_VEL
LIN {X 0,Y 300.224,Z 335.841,A -85,B 0,C 180,E1 -17511.444,E2 -17511.444} C_VEL
LIN {X 0,Y 308.534,Z 353.337,A -85,B 0,C 180,E1 -17513.178,E2 -17513.178} C_VEL
LIN {X 0,Y 304.254,Z 457.388,A -85,B 0,C 180,E1 -17515.582,E2 -17515.582} C_VEL
LIN {X 0,Y 303.102,Z 472.186,A -85,B 0,C 180,E1 -17516.136,E2 -17516.136} C_VEL
LIN {X 0,Y 301.61,Z 485.882,A -85,B 0,C 180,E1 -17516.877,E2 -17516.877} C_VEL
LIN {X 0,Y 299.547,Z 500.65,A -85,B 0,C 180,E1 -17517.946,E2 -17517.946} C_VEL
LIN {X 0,Y 297.158,Z 514.511,A -85,B 0,C 180,E1 -17519.239,E2 -17519.239} C_VEL
LIN {X 0,Y 294.545,Z 527.26,A -85,B 0,C 180,E1 -17520.715,E2 -17520.715} C_VEL
LIN {X 0,Y 291.451,Z 540.106,A -85,B 0,C 180,E1 -17522.536,E2 -17522.536} C_VEL
LIN {X 0,Y 288.653,Z 551.66,A -85,B 0,C 180,E1 -17524.575,E2 -17524.575} C_VEL
LIN {X 0,Y 285.738,Z 562.218,A -85,B 0,C 180,E1 -17526.825,E2 -17526.825} C_VEL
LIN {X 0,Y 283.137,Z 571.638,A -85,B 0,C 180,E1 -17529.285,E2 -17529.285} C_VEL
LIN {X 0,Y 280.867,Z 579.479,A -85,B 0,C 180,E1 -17531.773,E2 -17531.773} C_VEL
LIN {X 0,Y 278.983,Z 586.782,A -85,B 0,C 180,E1 -17534.661,E2 -17534.661} C_VEL
LIN {X 0,Y 277.395,Z 592.579,A -85,B 0,C 180,E1 -17537.563,E2 -17537.563} C_VEL
LIN {X 0,Y 276.622,Z 596.005,A -85,B 0,C 180,E1 -17539.755,E2 -17539.755} C_VEL
LIN {X 0,Y 275.92,Z 599.471,A -85,B 0,C 180,E1 -17542.682,E2 -17542.682} C_VEL
LIN {X 0,Y 275.559,Z 601.759,A -85,B 0,C 180,E1 -17545.611,E2 -17545.611} C_VEL
LIN {X 0,Y 275.355,Z 602.928,A -85,B 0,C 180,E1 -17548.537,E2 -17548.537} C_VEL
LIN {X 0,Y 275.354,Z 602.941,A -85,B 0,C 180,E1 -17551.462,E2 -17551.462} C_VEL
LIN {X 0,Y 275.558,Z 601.827,A -85,B 0,C 180,E1 -17554.388,E2 -17554.388} C_VEL
LIN {X 0,Y 275.919,Z 599.591,A -85,B 0,C 180,E1 -17557.316,E2 -17557.316} C_VEL
LIN {X 0,Y 276.612,Z 596.173,A -85,B 0,C 180,E1 -17560.244,E2 -17560.244} C_VEL
LIN {X 0,Y 277.652,Z 591.491,A -85,B 0,C 180,E1 -17563.168,E2 -17563.168} C_VEL
LIN {X 0,Y 279.347,Z 585.411,A -85,B 0,C 180,E1 -17566.065,E2 -17566.065} C_VEL
LIN {X 0,Y 281.409,Z 577.754,A -85,B 0,C 180,E1 -17568.945,E2 -17568.945} C_VEL
LIN {X 0,Y 283.733,Z 569.582,A -85,B 0,C 180,E1 -17571.429,E2 -17571.429} C_VEL
LIN {X 0,Y 286.515,Z 559.728,A -85,B 0,C 180,E1 -17573.874,E2 -17573.874} C_VEL
LIN {X 0,Y 289.128,Z 549.624,A -85,B 0,C 180,E1 -17575.946,E2 -17575.946} C_VEL
LIN {X 0,Y 292.197,Z 537.579,A -85,B 0,C 180,E1 -17577.97,E2 -17577.97} C_VEL
LIN {X 0,Y 294.958,Z 525.495,A -85,B 0,C 180,E1 -17579.63,E2 -17579.63} C_VEL
LIN {X 0,Y 297.619,Z 512.356,A -85,B 0,C 180,E1 -17581.101,E2 -17581.101} C_VEL
LIN {X 0,Y 300.038,Z 497.725,A -85,B 0,C 180,E1 -17582.411,E2 -17582.411} C_VEL
LIN {X 0,Y 302.002,Z 483.208,A -85,B 0,C 180,E1 -17583.402,E2 -17583.402} C_VEL
LIN {X 0,Y 303.543,Z 468.052,A -85,B 0,C 180,E1 -17584.157,E2 -17584.157} C_VEL
LIN {X 0,Y 304.605,Z 452.107,A -85,B 0,C 180,E1 -17584.672,E2 -17584.672} C_VEL
LIN {X 0,Y 308.666,Z 354.421,A -85,B 0,C 180,E1 -17586.897,E2 -17586.897} C_VEL
LIN {X 0,Y 308.294,Z 352.758,A -85,B 0,C 180,E1 -17586.997,E2 -17586.997} C_VEL
LIN {X 0,Y 300.462,Z 336.206,A -85,B 0,C 180,E1 -17588.637,E2 -17588.637} C_VEL
LIN {X 0,Y 295.284,Z 326.945,A -85,B 0,C 180,E1 -17589.739,E2 -17589.739} C_VEL
LIN {X 0,Y 285.452,Z 311.588,A -85,B 0,C 180,E1 -17591.924,E2 -17591.924} C_VEL
LIN {X 0,Y 282.263,Z 307.02,A -85,B 0,C 180,E1 -17592.668,E2 -17592.668} C_VEL
LIN {X 0,Y 280.174,Z 303.654,A -85,B 0,C 180,E1 -17593.183,E2 -17593.183} C_VEL
LIN {X 0,Y 278.384,Z 301.672,A -85,B 0,C 180,E1 -17593.602,E2 -17593.602} C_VEL
LIN {X 0,Y 276.892,Z 299.936,A -85,B 0,C 180,E1 -17594.062,E2 -17594.062} C_VEL
LIN {X 0,Y 275.055,Z 298.988,A -85,B 0,C 180,E1 -17594.816,E2 -17594.816} C_VEL
LIN {X 0,Y 272.434,Z 299.16,A -85,B 0,C 180,E1 -17596.367,E2 -17596.367} C_VEL
LIN {X 0,Y 270.724,Z 299.441,A -85,B 0,C 180,E1 -17598.13,E2 -17598.13} C_VEL
LIN {X 0,Y 270.109,Z 299.448,A -85,B 0,C 180,E1 -17599.934,E2 -17599.934} C_VEL
LIN {X 0,Y 270.212,Z 299.416,A -85,B 0,C 180,E1 -17603.734,E2 -17603.734} C_VEL
LIN {X 0,Y 270.199,Z 299.455,A -85,B 0,C 180,E1 -17606.892,E2 -17606.892} C_VEL
LIN {X 0,Y 270.154,Z 299.458,A -85,B 0,C 180,E1 -17610.377,E2 -17610.377} C_VEL
LIN {X 0,Y 270.175,Z 299.453,A -85,B 0,C 180,E1 -17613.754,E2 -17613.754} C_VEL
LIN {X 0,Y 270.179,Z 299.445,A -85,B 0,C 180,E1 -17617.034,E2 -17617.034} C_VEL
LIN {X 0,Y 270.217,Z 299.442,A -85,B 0,C 180,E1 -17620.238,E2 -17620.238} C_VEL
LIN {X 0,Y 270.336,Z 299.427,A -85,B 0,C 180,E1 -17624.931,E2 -17624.931} C_VEL
LIN {X 0,Y 270.407,Z 299.422,A -85,B 0,C 180,E1 -17629.517,E2 -17629.517} C_VEL
LIN {X 0,Y 270.559,Z 299.404,A -85,B 0,C 180,E1 -17632.537,E2 -17632.537} C_VEL
LIN {X 0,Y 270.772,Z 299.383,A -85,B 0,C 180,E1 -17638.513,E2 -17638.513} C_VEL
LIN {X 0,Y 270.775,Z 299.366,A -85,B 0,C 180,E1 -17641.487,E2 -17641.487} C_VEL
LIN {X 0,Y 270.561,Z 299.403,A -85,B 0,C 180,E1 -17647.462,E2 -17647.462} C_VEL
LIN {X 0,Y 270.408,Z 299.414,A -85,B 0,C 180,E1 -17650.482,E2 -17650.482} C_VEL
LIN {X 0,Y 270.401,Z 299.416,A -85,B 0,C 180,E1 -17655.065,E2 -17655.065} C_VEL
LIN {X 0,Y 270.3,Z 299.432,A -85,B 0,C 180,E1 -17659.755,E2 -17659.755} C_VEL
LIN {X 0,Y 270.224,Z 299.413,A -85,B 0,C 180,E1 -17664.59,E2 -17664.59} C_VEL
LIN {X 0,Y 270.2,Z 299.447,A -85,B 0,C 180,E1 -17667.916,E2 -17667.916} C_VEL
LIN {X 0,Y 270.171,Z 299.426,A -85,B 0,C 180,E1 -17671.35,E2 -17671.35} C_VEL
LIN {X 0,Y 270.199,Z 299.453,A -85,B 0,C 180,E1 -17674.906,E2 -17674.906} C_VEL
LIN {X 0,Y 270.195,Z 299.436,A -85,B 0,C 180,E1 -17678.711,E2 -17678.711} C_VEL
LIN {X 0,Y 270.179,Z 299.496,A -85,B 0,C 180,E1 -17681.108,E2 -17681.108} C_VEL
LIN {X 0,Y 273.491,Z 309.739,A -85,B 0,C 180,E1 -17685.206,E2 -17685.206} C_VEL
LIN {X 0,Y 276.432,Z 314.559,A -85,B 0,C 180,E1 -17685.974,E2 -17685.974} C_VEL
LIN {X 0,Y 283.295,Z 326.522,A -85,B 0,C 180,E1 -17687.691,E2 -17687.691} C_VEL
LIN {X 0,Y 291.201,Z 341.395,A -85,B 0,C 180,E1 -17689.551,E2 -17689.551} C_VEL
LIN {X 0,Y 299.308,Z 359.277,A -85,B 0,C 180,E1 -17691.389,E2 -17691.389} C_VEL
LIN {X 0,Y 301.094,Z 363.812,A -85,B 0,C 180,E1 -17691.792,E2 -17691.792} C_VEL
LIN {X 0,Y 302.309,Z 373.474,A -85,B 0,C 180,E1 -17692.255,E2 -17692.255} C_VEL
LIN {X 0,Y 298.079,Z 472.58,A -85,B 0,C 180,E1 -17694.56,E2 -17694.56} C_VEL
LIN {X 0,Y 296.916,Z 487.913,A -85,B 0,C 180,E1 -17695.075,E2 -17695.075} C_VEL
LIN {X 0,Y 295.162,Z 502.182,A -85,B 0,C 180,E1 -17695.77,E2 -17695.77} C_VEL
LIN {X 0,Y 292.938,Z 516.385,A -85,B 0,C 180,E1 -17696.716,E2 -17696.716} C_VEL
LIN {X 0,Y 290.348,Z 530.137,A -85,B 0,C 180,E1 -17697.907,E2 -17697.907} C_VEL
LIN {X 0,Y 287.56,Z 543.073,A -85,B 0,C 180,E1 -17699.324,E2 -17699.324} C_VEL
LIN {X 0,Y 284.221,Z 556.653,A -85,B 0,C 180,E1 -17701.173,E2 -17701.173} C_VEL
LIN {X 0,Y 280.938,Z 568.881,A -85,B 0,C 180,E1 -17703.238,E2 -17703.238} C_VEL
LIN {X 0,Y 278.182,Z 579,A -85,B 0,C 180,E1 -17705.326,E2 -17705.326} C_VEL
LIN {X 0,Y 275.375,Z 589.21,A -85,B 0,C 180,E1 -17707.887,E2 -17707.887} C_VEL
LIN {X 0,Y 272.992,Z 597.563,A -85,B 0,C 180,E1 -17710.448,E2 -17710.448} C_VEL
LIN {X 0,Y 270.954,Z 605.423,A -85,B 0,C 180,E1 -17713.423,E2 -17713.423} C_VEL
LIN {X 0,Y 269.559,Z 611.688,A -85,B 0,C 180,E1 -17716.43,E2 -17716.43} C_VEL
LIN {X 0,Y 268.648,Z 616.54,A -85,B 0,C 180,E1 -17719.449,E2 -17719.449} C_VEL
LIN {X 0,Y 268.271,Z 620.105,A -85,B 0,C 180,E1 -17722.474,E2 -17722.474} C_VEL
LIN {X 0,Y 268.154,Z 622.453,A -85,B 0,C 180,E1 -17725.491,E2 -17725.491} C_VEL
LIN {X 0,Y 268.224,Z 623.637,A -85,B 0,C 180,E1 -17728.499,E2 -17728.499} C_VEL
LIN {X 0,Y 268.224,Z 623.633,A -85,B 0,C 180,E1 -17731.502,E2 -17731.502} C_VEL
LIN {X 0,Y 268.154,Z 622.434,A -85,B 0,C 180,E1 -17734.51,E2 -17734.51} C_VEL
LIN {X 0,Y 268.251,Z 620.071,A -85,B 0,C 180,E1 -17737.528,E2 -17737.528} C_VEL
LIN {X 0,Y 268.644,Z 616.499,A -85,B 0,C 180,E1 -17740.553,E2 -17740.553} C_VEL
LIN {X 0,Y 269.56,Z 611.635,A -85,B 0,C 180,E1 -17743.572,E2 -17743.572} C_VEL
LIN {X 0,Y 270.956,Z 605.347,A -85,B 0,C 180,E1 -17746.579,E2 -17746.579} C_VEL
LIN {X 0,Y 272.972,Z 597.465,A -85,B 0,C 180,E1 -17749.555,E2 -17749.555} C_VEL
LIN {X 0,Y 275.361,Z 589.098,A -85,B 0,C 180,E1 -17752.116,E2 -17752.116} C_VEL
LIN {X 0,Y 278.148,Z 578.953,A -85,B 0,C 180,E1 -17754.657,E2 -17754.657} C_VEL
LIN {X 0,Y 280.938,Z 568.731,A -85,B 0,C 180,E1 -17756.763,E2 -17756.763} C_VEL
LIN {X 0,Y 284.198,Z 556.475,A -85,B 0,C 180,E1 -17758.831,E2 -17758.831} C_VEL
LIN {X 0,Y 287.247,Z 544.182,A -85,B 0,C 180,E1 -17760.511,E2 -17760.511} C_VEL
LIN {X 0,Y 290.072,Z 531.152,A -85,B 0,C 180,E1 -17761.961,E2 -17761.961} C_VEL
LIN {X 0,Y 292.556,Z 518.026,A -85,B 0,C 180,E1 -17763.129,E2 -17763.129} C_VEL
LIN {X 0,Y 294.775,Z 504.344,A -85,B 0,C 180,E1 -17764.076,E2 -17764.076} C_VEL
LIN {X 0,Y 296.7,Z 489.113,A -85,B 0,C 180,E1 -17764.853,E2 -17764.853} C_VEL
LIN {X 0,Y 297.967,Z 473.017,A -85,B 0,C 180,E1 -17765.405,E2 -17765.405} C_VEL
LIN {X 0,Y 301.432,Z 391.201,A -85,B 0,C 180,E1 -17767.316,E2 -17767.316} C_VEL
LIN {X 0,Y 302.219,Z 372.394,A -85,B 0,C 180,E1 -17767.753,E2 -17767.753} C_VEL
LIN {X 0,Y 300.689,Z 362.766,A -85,B 0,C 180,E1 -17768.262,E2 -17768.262} C_VEL
LIN {X 0,Y 293.117,Z 345.43,A -85,B 0,C 180,E1 -17769.965,E2 -17769.965} C_VEL
LIN {X 0,Y 284.317,Z 328.285,A -85,B 0,C 180,E1 -17772.018,E2 -17772.018} C_VEL
LIN {X 0,Y 276.176,Z 314.213,A -85,B 0,C 180,E1 -17774.037,E2 -17774.037} C_VEL
LIN {X 0,Y 273.349,Z 309.421,A -85,B 0,C 180,E1 -17774.815,E2 -17774.815} C_VEL
LIN {X 0,Y 271.106,Z 302.389,A -85,B 0,C 180,E1 -17777.623,E2 -17777.623} C_VEL
LIN {X 0,Y 270.178,Z 299.455,A -85,B 0,C 180,E1 -17778.892,E2 -17778.892} C_VEL
LIN {X 0,Y 270.21,Z 299.449,A -85,B 0,C 180,E1 -17781.375,E2 -17781.375} C_VEL
LIN {X 0,Y 270.205,Z 299.444,A -85,B 0,C 180,E1 -17785.095,E2 -17785.095} C_VEL
LIN {X 0,Y 270.187,Z 299.45,A -85,B 0,C 180,E1 -17789.137,E2 -17789.137} C_VEL
LIN {X 0,Y 270.226,Z 299.447,A -85,B 0,C 180,E1 -17792.163,E2 -17792.163} C_VEL
LIN {X 0,Y 270.232,Z 299.446,A -85,B 0,C 180,E1 -17795.543,E2 -17795.543} C_VEL
LIN {X 0,Y 270.304,Z 299.432,A -85,B 0,C 180,E1 -17800.245,E2 -17800.245} C_VEL
LIN {X 0,Y 270.408,Z 299.417,A -85,B 0,C 180,E1 -17804.936,E2 -17804.936} C_VEL
LIN {X 0,Y 270.415,Z 299.418,A -85,B 0,C 180,E1 -17809.518,E2 -17809.518} C_VEL
LIN {X 0,Y 270.567,Z 299.396,A -85,B 0,C 180,E1 -17812.538,E2 -17812.538} C_VEL
LIN {X 0,Y 270.78,Z 299.377,A -85,B 0,C 180,E1 -17818.513,E2 -17818.513} C_VEL
LIN {X 0,Y 270.776,Z 299.371,A -85,B 0,C 180,E1 -17821.487,E2 -17821.487} C_VEL
LIN {X 0,Y 270.566,Z 299.403,A -85,B 0,C 180,E1 -17827.463,E2 -17827.463} C_VEL
LIN {X 0,Y 270.392,Z 299.417,A -85,B 0,C 180,E1 -17830.483,E2 -17830.483} C_VEL
LIN {X 0,Y 270.343,Z 299.424,A -85,B 0,C 180,E1 -17835.068,E2 -17835.068} C_VEL
LIN {X 0,Y 270.223,Z 299.444,A -85,B 0,C 180,E1 -17839.762,E2 -17839.762} C_VEL
LIN {X 0,Y 270.188,Z 299.454,A -85,B 0,C 180,E1 -17844.437,E2 -17844.437} C_VEL
LIN {X 0,Y 270.188,Z 299.421,A -85,B 0,C 180,E1 -17847.918,E2 -17847.918} C_VEL
LIN {X 0,Y 270.173,Z 299.458,A -85,B 0,C 180,E1 -17851.35,E2 -17851.35} C_VEL
LIN {X 0,Y 270.201,Z 299.452,A -85,B 0,C 180,E1 -17854.906,E2 -17854.906} C_VEL
LIN {X 0,Y 270.201,Z 299.445,A -85,B 0,C 180,E1 -17858.71,E2 -17858.71} C_VEL
LIN {X 0,Y 270.124,Z 299.458,A -85,B 0,C 180,E1 -17863.238,E2 -17863.238} C_VEL
LIN {X 0,Y 270.121,Z 299.46,A -85,B 0,C 180,E1 -17864.743,E2 -17864.743} C_VEL
LIN {X 0,Y 271.04,Z 302.173,A -85,B 0,C 180,E1 -17865.053,E2 -17865.053} C_VEL
LIN {X 0,Y 273.317,Z 304.824,A -85,B 0,C 180,E1 -17865.629,E2 -17865.629} C_VEL
LIN {X 0,Y 275.548,Z 308.274,A -85,B 0,C 180,E1 -17866.208,E2 -17866.208} C_VEL
LIN {X 0,Y 280.302,Z 315.219,A -85,B 0,C 180,E1 -17867.38,E2 -17867.38} C_VEL
LIN {X 0,Y 288.937,Z 328.429,A -85,B 0,C 180,E1 -17869.379,E2 -17869.379} C_VEL
LIN {X 0,Y 295.04,Z 339.111,A -85,B 0,C 180,E1 -17870.73,E2 -17870.73} C_VEL
LIN {X 0,Y 302.853,Z 355.664,A -85,B 0,C 180,E1 -17872.429,E2 -17872.429} C_VEL
LIN {X 0,Y 298.363,Z 459.091,A -85,B 0,C 180,E1 -17874.855,E2 -17874.855} C_VEL
LIN {X 0,Y 297.054,Z 474.352,A -85,B 0,C 180,E1 -17875.458,E2 -17875.458} C_VEL
LIN {X 0,Y 295.417,Z 488.494,A -85,B 0,C 180,E1 -17876.275,E2 -17876.275} C_VEL
LIN {X 0,Y 293.221,Z 503.184,A -85,B 0,C 180,E1 -17877.402,E2 -17877.402} C_VEL
LIN {X 0,Y 290.464,Z 517.915,A -85,B 0,C 180,E1 -17878.856,E2 -17878.856} C_VEL
LIN {X 0,Y 287.492,Z 531.351,A -85,B 0,C 180,E1 -17880.529,E2 -17880.529} C_VEL
LIN {X 0,Y 284.367,Z 543.543,A -85,B 0,C 180,E1 -17882.393,E2 -17882.393} C_VEL
LIN {X 0,Y 281.47,Z 554.937,A -85,B 0,C 180,E1 -17884.558,E2 -17884.558} C_VEL
LIN {X 0,Y 278.413,Z 565.407,A -85,B 0,C 180,E1 -17886.966,E2 -17886.966} C_VEL
LIN {X 0,Y 275.738,Z 574.345,A -85,B 0,C 180,E1 -17889.484,E2 -17889.484} C_VEL
LIN {X 0,Y 273.503,Z 581.745,A -85,B 0,C 180,E1 -17892.039,E2 -17892.039} C_VEL
LIN {X 0,Y 271.632,Z 588.651,A -85,B 0,C 180,E1 -17895.004,E2 -17895.004} C_VEL
LIN {X 0,Y 270.129,Z 594.076,A -85,B 0,C 180,E1 -17897.986,E2 -17897.986} C_VEL
LIN {X 0,Y 269.187,Z 598.162,A -85,B 0,C 180,E1 -17900.987,E2 -17900.987} C_VEL
LIN {X 0,Y 268.649,Z 601.029,A -85,B 0,C 180,E1 -17903.993,E2 -17903.993} C_VEL
LIN {X 0,Y 268.387,Z 602.751,A -85,B 0,C 180,E1 -17906.997,E2 -17906.997} C_VEL
LIN {X 0,Y 268.261,Z 603.353,A -85,B 0,C 180,E1 -17909.999,E2 -17909.999} C_VEL
LIN {X 0,Y 268.386,Z 602.791,A -85,B 0,C 180,E1 -17913.001,E2 -17913.001} C_VEL
LIN {X 0,Y 268.669,Z 600.934,A -85,B 0,C 180,E1 -17916.264,E2 -17916.264} C_VEL
LIN {X 0,Y 269.183,Z 598.305,A -85,B 0,C 180,E1 -17919.012,E2 -17919.012} C_VEL
LIN {X 0,Y 270.095,Z 594.268,A -85,B 0,C 180,E1 -17922.014,E2 -17922.014} C_VEL
LIN {X 0,Y 271.583,Z 588.904,A -85,B 0,C 180,E1 -17924.997,E2 -17924.997} C_VEL
LIN {X 0,Y 273.454,Z 582.068,A -85,B 0,C 180,E1 -17927.963,E2 -17927.963} C_VEL
LIN {X 0,Y 276.037,Z 573.52,A -85,B 0,C 180,E1 -17930.881,E2 -17930.881} C_VEL
LIN {X 0,Y 278.699,Z 564.428,A -85,B 0,C 180,E1 -17933.401,E2 -17933.401} C_VEL
LIN {X 0,Y 281.628,Z 554.44,A -85,B 0,C 180,E1 -17935.666,E2 -17935.666} C_VEL
LIN {X 0,Y 284.551,Z 543.158,A -85,B 0,C 180,E1 -17937.786,E2 -17937.786} C_VEL
LIN {X 0,Y 287.697,Z 530.887,A -85,B 0,C 180,E1 -17939.648,E2 -17939.648} C_VEL
LIN {X 0,Y 290.364,Z 518.803,A -85,B 0,C 180,E1 -17941.155,E2 -17941.155} C_VEL
LIN {X 0,Y 292.666,Z 506.641,A -85,B 0,C 180,E1 -17942.401,E2 -17942.401} C_VEL
LIN {X 0,Y 294.759,Z 493.733,A -85,B 0,C 180,E1 -17943.467,E2 -17943.467} C_VEL
LIN {X 0,Y 296.681,Z 478.732,A -85,B 0,C 180,E1 -17944.42,E2 -17944.42} C_VEL
LIN {X 0,Y 298.033,Z 464.177,A -85,B 0,C 180,E1 -17945.085,E2 -17945.085} C_VEL
LIN {X 0,Y 299.102,Z 447.188,A -85,B 0,C 180,E1 -17945.559,E2 -17945.559} C_VEL
LIN {X 0,Y 302.877,Z 355.624,A -85,B 0,C 180,E1 -17947.696,E2 -17947.696} C_VEL
LIN {X 0,Y 294.992,Z 338.91,A -85,B 0,C 180,E1 -17949.415,E2 -17949.415} C_VEL
LIN {X 0,Y 287.88,Z 326.829,A -85,B 0,C 180,E1 -17950.99,E2 -17950.99} C_VEL
LIN {X 0,Y 280.73,Z 315.797,A -85,B 0,C 180,E1 -17952.658,E2 -17952.658} C_VEL
LIN {X 0,Y 275.58,Z 308.247,A -85,B 0,C 180,E1 -17953.93,E2 -17953.93} C_VEL
LIN {X 0,Y 273.388,Z 304.898,A -85,B 0,C 180,E1 -17954.499,E2 -17954.499} C_VEL
LIN {X 0,Y 270.881,Z 301.825,A -85,B 0,C 180,E1 -17955.14,E2 -17955.14} C_VEL
LIN {X 0,Y 270.146,Z 299.461,A -85,B 0,C 180,E1 -17955.426,E2 -17955.426} C_VEL
LIN {X 0,Y 270.127,Z 299.446,A -85,B 0,C 180,E1 -17959.425,E2 -17959.425} C_VEL
LIN {X 0,Y 270.109,Z 299.448,A -85,B 0,C 180,E1 -17959.934,E2 -17959.934} C_VEL
LIN {X 0,Y 269.447,Z 299.544,A -85,B 0,C 180,E1 -17961.179,E2 -17961.179} C_VEL
LIN {X 0,Y 266.635,Z 299.882,A -85,B 0,C 180,E1 -17963.21,E2 -17963.21} C_VEL
LIN {X 0,Y 264.242,Z 300.18,A -85,B 0,C 180,E1 -17964.861,E2 -17964.861} C_VEL
LIN {X 0,Y 263.201,Z 300.318,A -85,B 0,C 180,E1 -17966.139,E2 -17966.139} C_VEL
LIN {X 0,Y 263.109,Z 300.323,A -85,B 0,C 180,E1 -17966.572,E2 -17966.572} C_VEL
LIN {X 0,Y 263.107,Z 300.33,A -85,B 0,C 180,E1 -17969.501,E2 -17969.501} C_VEL
LIN {X 0,Y 263.11,Z 300.327,A -85,B 0,C 180,E1 -17972.993,E2 -17972.993} C_VEL
LIN {X 0,Y 263.113,Z 300.325,A -85,B 0,C 180,E1 -17976.38,E2 -17976.38} C_VEL
LIN {X 0,Y 263.205,Z 300.322,A -85,B 0,C 180,E1 -17979.688,E2 -17979.688} C_VEL
LIN {X 0,Y 263.286,Z 300.309,A -85,B 0,C 180,E1 -17984.518,E2 -17984.518} C_VEL
LIN {X 0,Y 263.345,Z 300.304,A -85,B 0,C 180,E1 -17989.233,E2 -17989.233} C_VEL
LIN {X 0,Y 263.524,Z 300.278,A -85,B 0,C 180,E1 -17992.337,E2 -17992.337} C_VEL
LIN {X 0,Y 263.736,Z 300.259,A -85,B 0,C 180,E1 -17998.473,E2 -17998.473} C_VEL
LIN {X 0,Y 263.738,Z 300.242,A -85,B 0,C 180,E1 -18001.527,E2 -18001.527} C_VEL
LIN {X 0,Y 263.525,Z 300.281,A -85,B 0,C 180,E1 -18007.663,E2 -18007.663} C_VEL
LIN {X 0,Y 263.351,Z 300.292,A -85,B 0,C 180,E1 -18010.766,E2 -18010.766} C_VEL
LIN {X 0,Y 263.349,Z 300.295,A -85,B 0,C 180,E1 -18015.478,E2 -18015.478} C_VEL
LIN {X 0,Y 263.266,Z 300.311,A -85,B 0,C 180,E1 -18020.306,E2 -18020.306} C_VEL
LIN {X 0,Y 263.167,Z 300.289,A -85,B 0,C 180,E1 -18025.295,E2 -18025.295} C_VEL
LIN {X 0,Y 263.133,Z 300.334,A -85,B 0,C 180,E1 -18028.735,E2 -18028.735} C_VEL
LIN {X 0,Y 263.126,Z 300.302,A -85,B 0,C 180,E1 -18032.289,E2 -18032.289} C_VEL
LIN {X 0,Y 263.179,Z 300.304,A -85,B 0,C 180,E1 -18036.763,E2 -18036.763} C_VEL
LIN {X 0,Y 263.105,Z 300.345,A -85,B 0,C 180,E1 -18039.776,E2 -18039.776} C_VEL
LIN {X 0,Y 266.017,Z 309.233,A -85,B 0,C 180,E1 -18043.58,E2 -18043.58} C_VEL
LIN {X 0,Y 268.956,Z 314.04,A -85,B 0,C 180,E1 -18044.408,E2 -18044.408} C_VEL
LIN {X 0,Y 276.024,Z 325.891,A -85,B 0,C 180,E1 -18046.292,E2 -18046.292} C_VEL
LIN {X 0,Y 282.968,Z 338.603,A -85,B 0,C 180,E1 -18048.035,E2 -18048.035} C_VEL
LIN {X 0,Y 289.848,Z 352.707,A -85,B 0,C 180,E1 -18049.685,E2 -18049.685} C_VEL
LIN {X 0,Y 295.689,Z 366.336,A -85,B 0,C 180,E1 -18051.047,E2 -18051.047} C_VEL
LIN {X 0,Y 296.645,Z 374.573,A -85,B 0,C 180,E1 -18051.444,E2 -18051.444} C_VEL
LIN {X 0,Y 292.794,Z 462.099,A -85,B 0,C 180,E1 -18053.5,E2 -18053.5} C_VEL
LIN {X 0,Y 291.688,Z 481.481,A -85,B 0,C 180,E1 -18054.035,E2 -18054.035} C_VEL
LIN {X 0,Y 290.039,Z 496.874,A -85,B 0,C 180,E1 -18054.707,E2 -18054.707} C_VEL
LIN {X 0,Y 287.763,Z 511.733,A -85,B 0,C 180,E1 -18055.614,E2 -18055.614} C_VEL
LIN {X 0,Y 285.225,Z 525.668,A -85,B 0,C 180,E1 -18056.754,E2 -18056.754} C_VEL
LIN {X 0,Y 282.296,Z 539.344,A -85,B 0,C 180,E1 -18058.182,E2 -18058.182} C_VEL
LIN {X 0,Y 279.212,Z 551.705,A -85,B 0,C 180,E1 -18059.774,E2 -18059.774} C_VEL
LIN {X 0,Y 276.261,Z 562.776,A -85,B 0,C 180,E1 -18061.511,E2 -18061.511} C_VEL
LIN {X 0,Y 273.028,Z 573.968,A -85,B 0,C 180,E1 -18063.639,E2 -18063.639} C_VEL
LIN {X 0,Y 269.876,Z 584.841,A -85,B 0,C 180,E1 -18066.195,E2 -18066.195} C_VEL
LIN {X 0,Y 267.206,Z 593.906,A -85,B 0,C 180,E1 -18068.799,E2 -18068.799} C_VEL
LIN {X 0,Y 265.064,Z 601.435,A -85,B 0,C 180,E1 -18071.448,E2 -18071.448} C_VEL
LIN {X 0,Y 263.241,Z 608.469,A -85,B 0,C 180,E1 -18074.516,E2 -18074.516} C_VEL
LIN {X 0,Y 262.028,Z 614.009,A -85,B 0,C 180,E1 -18077.61,E2 -18077.61} C_VEL
LIN {X 0,Y 261.322,Z 618.205,A -85,B 0,C 180,E1 -18080.715,E2 -18080.715} C_VEL
LIN {X 0,Y 261.133,Z 621.157,A -85,B 0,C 180,E1 -18083.821,E2 -18083.821} C_VEL
LIN {X 0,Y 261.1,Z 622.919,A -85,B 0,C 180,E1 -18086.915,E2 -18086.915} C_VEL
LIN {X 0,Y 261.175,Z 623.523,A -85,B 0,C 180,E1 -18090.001,E2 -18090.001} C_VEL
LIN {X 0,Y 261.1,Z 622.907,A -85,B 0,C 180,E1 -18093.087,E2 -18093.087} C_VEL
LIN {X 0,Y 261.13,Z 621.13,A -85,B 0,C 180,E1 -18096.181,E2 -18096.181} C_VEL
LIN {X 0,Y 261.321,Z 618.167,A -85,B 0,C 180,E1 -18099.287,E2 -18099.287} C_VEL
LIN {X 0,Y 262.025,Z 613.962,A -85,B 0,C 180,E1 -18102.391,E2 -18102.391} C_VEL
LIN {X 0,Y 263.244,Z 608.403,A -85,B 0,C 180,E1 -18105.485,E2 -18105.485} C_VEL
LIN {X 0,Y 265.065,Z 601.344,A -85,B 0,C 180,E1 -18108.553,E2 -18108.553} C_VEL
LIN {X 0,Y 267.542,Z 592.575,A -85,B 0,C 180,E1 -18111.579,E2 -18111.579} C_VEL
LIN {X 0,Y 269.904,Z 584.727,A -85,B 0,C 180,E1 -18113.804,E2 -18113.804} C_VEL
LIN {X 0,Y 273.032,Z 573.822,A -85,B 0,C 180,E1 -18116.362,E2 -18116.362} C_VEL
LIN {X 0,Y 276.498,Z 561.575,A -85,B 0,C 180,E1 -18118.671,E2 -18118.671} C_VEL
LIN {X 0,Y 279.833,Z 549.096,A -85,B 0,C 180,E1 -18120.57,E2 -18120.57} C_VEL
LIN {X 0,Y 283.1,Z 535.507,A -85,B 0,C 180,E1 -18122.231,E2 -18122.231} C_VEL
LIN {X 0,Y 285.882,Z 521.73,A -85,B 0,C 180,E1 -18123.583,E2 -18123.583} C_VEL
LIN {X 0,Y 288.477,Z 506.667,A -85,B 0,C 180,E1 -18124.714,E2 -18124.714} C_VEL
LIN {X 0,Y 290.62,Z 491.585,A -85,B 0,C 180,E1 -18125.532,E2 -18125.532} C_VEL
LIN {X 0,Y 292.038,Z 475.745,A -85,B 0,C 180,E1 -18126.13,E2 -18126.13} C_VEL
LIN {X 0,Y 295.731,Z 393.577,A -85,B 0,C 180,E1 -18128.082,E2 -18128.082} C_VEL
LIN {X 0,Y 296.579,Z 373.61,A -85,B 0,C 180,E1 -18128.556,E2 -18128.556} C_VEL
LIN {X 0,Y 295.282,Z 365.549,A -85,B 0,C 180,E1 -18129.001,E2 -18129.001} C_VEL
LIN {X 0,Y 288.185,Z 349.207,A -85,B 0,C 180,E1 -18130.662,E2 -18130.662} C_VEL
LIN {X 0,Y 280.109,Z 333.162,A -85,B 0,C 180,E1 -18132.625,E2 -18132.625} C_VEL
LIN {X 0,Y 272.075,Z 319.103,A -85,B 0,C 180,E1 -18134.692,E2 -18134.692} C_VEL
LIN {X 0,Y 268.401,Z 313.314,A -85,B 0,C 180,E1 -18135.681,E2 -18135.681} C_VEL
LIN {X 0,Y 265.981,Z 309.01,A -85,B 0,C 180,E1 -18136.418,E2 -18136.418} C_VEL
LIN {X 0,Y 263.11,Z 300.332,A -85,B 0,C 180,E1 -18140.224,E2 -18140.224} C_VEL
LIN {X 0,Y 263.166,Z 300.323,A -85,B 0,C 180,E1 -18144.019,E2 -18144.019} C_VEL
LIN {X 0,Y 263.131,Z 300.322,A -85,B 0,C 180,E1 -18147.712,E2 -18147.712} C_VEL
LIN {X 0,Y 263.152,Z 300.325,A -85,B 0,C 180,E1 -18151.805,E2 -18151.805} C_VEL
LIN {X 0,Y 263.194,Z 300.322,A -85,B 0,C 180,E1 -18155.218,E2 -18155.218} C_VEL
LIN {X 0,Y 263.267,Z 300.314,A -85,B 0,C 180,E1 -18159.694,E2 -18159.694} C_VEL
LIN {X 0,Y 263.356,Z 300.296,A -85,B 0,C 180,E1 -18164.522,E2 -18164.522} C_VEL
LIN {X 0,Y 263.358,Z 300.295,A -85,B 0,C 180,E1 -18169.234,E2 -18169.234} C_VEL
LIN {X 0,Y 263.531,Z 300.274,A -85,B 0,C 180,E1 -18172.337,E2 -18172.337} C_VEL
LIN {X 0,Y 263.743,Z 300.253,A -85,B 0,C 180,E1 -18178.473,E2 -18178.473} C_VEL
LIN {X 0,Y 263.74,Z 300.247,A -85,B 0,C 180,E1 -18181.527,E2 -18181.527} C_VEL
LIN {X 0,Y 263.53,Z 300.281,A -85,B 0,C 180,E1 -18187.663,E2 -18187.663} C_VEL
LIN {X 0,Y 263.337,Z 300.296,A -85,B 0,C 180,E1 -18190.767,E2 -18190.767} C_VEL
LIN {X 0,Y 263.292,Z 300.304,A -85,B 0,C 180,E1 -18195.482,E2 -18195.482} C_VEL
LIN {X 0,Y 263.211,Z 300.324,A -85,B 0,C 180,E1 -18200.311,E2 -18200.311} C_VEL
LIN {X 0,Y 263.125,Z 300.331,A -85,B 0,C 180,E1 -18205.3,E2 -18205.3} C_VEL
LIN {X 0,Y 263.121,Z 300.302,A -85,B 0,C 180,E1 -18208.737,E2 -18208.737} C_VEL
LIN {X 0,Y 263.13,Z 300.33,A -85,B 0,C 180,E1 -18212.289,E2 -18212.289} C_VEL
LIN {X 0,Y 263.177,Z 300.323,A -85,B 0,C 180,E1 -18216.76,E2 -18216.76} C_VEL
LIN {X 0,Y 263.093,Z 300.336,A -85,B 0,C 180,E1 -18219.875,E2 -18219.875} C_VEL
LIN {X 0,Y 263.113,Z 300.479,A -85,B 0,C 180,E1 -18223.218,E2 -18223.218} C_VEL
LIN {X 0,Y 263.978,Z 303.038,A -85,B 0,C 180,E1 -18223.52,E2 -18223.52} C_VEL
LIN {X 0,Y 266.03,Z 305.276,A -85,B 0,C 180,E1 -18224.073,E2 -18224.073} C_VEL
LIN {X 0,Y 268.516,Z 309.108,A -85,B 0,C 180,E1 -18224.768,E2 -18224.768} C_VEL
LIN {X 0,Y 269.909,Z 310.996,A -85,B 0,C 180,E1 -18225.138,E2 -18225.138} C_VEL
LIN {X 0,Y 277.893,Z 322.616,A -85,B 0,C 180,E1 -18227.174,E2 -18227.174} C_VEL
LIN {X 0,Y 286.305,Z 336.14,A -85,B 0,C 180,E1 -18229.173,E2 -18229.173} C_VEL
LIN {X 0,Y 291.148,Z 344.988,A -85,B 0,C 180,E1 -18230.28,E2 -18230.28} C_VEL
LIN {X 0,Y 297.149,Z 357.921,A -85,B 0,C 180,E1 -18231.637,E2 -18231.637} C_VEL
LIN {X 0,Y 292.609,Z 459.377,A -85,B 0,C 180,E1 -18234.058,E2 -18234.058} C_VEL
LIN {X 0,Y 291.254,Z 474.632,A -85,B 0,C 180,E1 -18234.668,E2 -18234.668} C_VEL
LIN {X 0,Y 289.406,Z 489.889,A -85,B 0,C 180,E1 -18235.572,E2 -18235.572} C_VEL
LIN {X 0,Y 287.215,Z 503.803,A -85,B 0,C 180,E1 -18236.669,E2 -18236.669} C_VEL
LIN {X 0,Y 284.428,Z 518.189,A -85,B 0,C 180,E1 -18238.118,E2 -18238.118} C_VEL
LIN {X 0,Y 281.337,Z 531.625,A -85,B 0,C 180,E1 -18239.818,E2 -18239.818} C_VEL
LIN {X 0,Y 278.08,Z 543.817,A -85,B 0,C 180,E1 -18241.713,E2 -18241.713} C_VEL
LIN {X 0,Y 275.028,Z 555.322,A -85,B 0,C 180,E1 -18243.945,E2 -18243.945} C_VEL
LIN {X 0,Y 271.878,Z 565.681,A -85,B 0,C 180,E1 -18246.379,E2 -18246.379} C_VEL
LIN {X 0,Y 269.092,Z 574.617,A -85,B 0,C 180,E1 -18248.953,E2 -18248.953} C_VEL
LIN {X 0,Y 266.734,Z 582.018,A -85,B 0,C 180,E1 -18251.567,E2 -18251.567} C_VEL
LIN {X 0,Y 264.774,Z 588.923,A -85,B 0,C 180,E1 -18254.606,E2 -18254.606} C_VEL
LIN {X 0,Y 263.164,Z 594.348,A -85,B 0,C 180,E1 -18257.663,E2 -18257.663} C_VEL
LIN {X 0,Y 262.162,Z 598.434,A -85,B 0,C 180,E1 -18260.743,E2 -18260.743} C_VEL
LIN {X 0,Y 261.592,Z 601.3,A -85,B 0,C 180,E1 -18263.83,E2 -18263.83} C_VEL
LIN {X 0,Y 261.321,Z 603.02,A -85,B 0,C 180,E1 -18266.916,E2 -18266.916} C_VEL
LIN {X 0,Y 261.185,Z 603.622,A -85,B 0,C 180,E1 -18269.999,E2 -18269.999} C_VEL
LIN {X 0,Y 261.321,Z 603.06,A -85,B 0,C 180,E1 -18273.083,E2 -18273.083} C_VEL
LIN {X 0,Y 261.59,Z 601.337,A -85,B 0,C 180,E1 -18276.247,E2 -18276.247} C_VEL
LIN {X 0,Y 262.158,Z 598.576,A -85,B 0,C 180,E1 -18279.255,E2 -18279.255} C_VEL
LIN {X 0,Y 263.133,Z 594.538,A -85,B 0,C 180,E1 -18282.337,E2 -18282.337} C_VEL
LIN {X 0,Y 264.717,Z 589.173,A -85,B 0,C 180,E1 -18285.395,E2 -18285.395} C_VEL
LIN {X 0,Y 266.694,Z 582.337,A -85,B 0,C 180,E1 -18288.434,E2 -18288.434} C_VEL
LIN {X 0,Y 269.398,Z 573.789,A -85,B 0,C 180,E1 -18291.421,E2 -18291.421} C_VEL
LIN {X 0,Y 272.177,Z 564.697,A -85,B 0,C 180,E1 -18293.996,E2 -18293.996} C_VEL
LIN {X 0,Y 275.136,Z 554.971,A -85,B 0,C 180,E1 -18296.255,E2 -18296.255} C_VEL
LIN {X 0,Y 278.268,Z 543.426,A -85,B 0,C 180,E1 -18298.47,E2 -18298.47} C_VEL
LIN {X 0,Y 281.538,Z 531.153,A -85,B 0,C 180,E1 -18300.364,E2 -18300.364} C_VEL
LIN {X 0,Y 284.321,Z 519.068,A -85,B 0,C 180,E1 -18301.894,E2 -18301.894} C_VEL
LIN {X 0,Y 286.924,Z 505.748,A -85,B 0,C 180,E1 -18303.27,E2 -18303.27} C_VEL
LIN {X 0,Y 289.069,Z 492.674,A -85,B 0,C 180,E1 -18304.34,E2 -18304.34} C_VEL
LIN {X 0,Y 290.957,Z 478.156,A -85,B 0,C 180,E1 -18305.255,E2 -18305.255} C_VEL
LIN {X 0,Y 292.381,Z 463.292,A -85,B 0,C 180,E1 -18305.919,E2 -18305.919} C_VEL
LIN {X 0,Y 293.431,Z 445.648,A -85,B 0,C 180,E1 -18306.408,E2 -18306.408} C_VEL
LIN {X 0,Y 297.261,Z 358.592,A -85,B 0,C 180,E1 -18308.454,E2 -18308.454} C_VEL
LIN {X 0,Y 296.725,Z 356.809,A -85,B 0,C 180,E1 -18308.591,E2 -18308.591} C_VEL
LIN {X 0,Y 289.751,Z 342.096,A -85,B 0,C 180,E1 -18310.178,E2 -18310.178} C_VEL
LIN {X 0,Y 281.687,Z 328.506,A -85,B 0,C 180,E1 -18312.047,E2 -18312.047} C_VEL
LIN {X 0,Y 273.678,Z 316.395,A -85,B 0,C 180,E1 -18314.025,E2 -18314.025} C_VEL
LIN {X 0,Y 271.139,Z 312.785,A -85,B 0,C 180,E1 -18314.682,E2 -18314.682} C_VEL
LIN {X 0,Y 268.976,Z 309.565,A -85,B 0,C 180,E1 -18315.264,E2 -18315.264} C_VEL
LIN {X 0,Y 266.622,Z 306.219,A -85,B 0,C 180,E1 -18315.908,E2 -18315.908} C_VEL
LIN {X 0,Y 265.853,Z 305.127,A -85,B 0,C 180,E1 -18316.123,E2 -18316.123} C_VEL
LIN {X 0,Y 263.922,Z 302.871,A -85,B 0,C 180,E1 -18316.652,E2 -18316.652} C_VEL
LIN {X 0,Y 263.111,Z 300.313,A -85,B 0,C 180,E1 -18316.971,E2 -18316.971} C_VEL
LIN {X 0,Y 263.088,Z 300.34,A -85,B 0,C 180,E1 -18320.776,E2 -18320.776} C_VEL
LIN {X 0,Y 263.151,Z 300.296,A -85,B 0,C 180,E1 -18324.016,E2 -18324.016} C_VEL
LIN {X 0,Y 263.109,Z 300.323,A -85,B 0,C 180,E1 -18326.572,E2 -18326.572} C_VEL
LIN {X 0,Y 262.415,Z 300.419,A -85,B 0,C 180,E1 -18327.85,E2 -18327.85} C_VEL
LIN {X 0,Y 259.543,Z 300.778,A -85,B 0,C 180,E1 -18329.933,E2 -18329.933} C_VEL
LIN {X 0,Y 257.13,Z 301.075,A -85,B 0,C 180,E1 -18331.627,E2 -18331.627} C_VEL
LIN {X 0,Y 256.114,Z 301.198,A -85,B 0,C 180,E1 -18332.94,E2 -18332.94} C_VEL
LIN {X 0,Y 256.041,Z 301.209,A -85,B 0,C 180,E1 -18333.385,E2 -18333.385} C_VEL
LIN {X 0,Y 256.055,Z 301.205,A -85,B 0,C 180,E1 -18337.402,E2 -18337.402} C_VEL
LIN {X 0,Y 256.103,Z 301.196,A -85,B 0,C 180,E1 -18340.773,E2 -18340.773} C_VEL
LIN {X 0,Y 256.21,Z 301.194,A -85,B 0,C 180,E1 -18344.079,E2 -18344.079} C_VEL
LIN {X 0,Y 256.285,Z 301.185,A -85,B 0,C 180,E1 -18348.933,E2 -18348.933} C_VEL
LIN {X 0,Y 256.466,Z 301.155,A -85,B 0,C 180,E1 -18352.125,E2 -18352.125} C_VEL
LIN {X 0,Y 256.459,Z 301.153,A -85,B 0,C 180,E1 -18356.858,E2 -18356.858} C_VEL
LIN {X 0,Y 256.698,Z 301.136,A -85,B 0,C 180,E1 -18358.431,E2 -18358.431} C_VEL
LIN {X 0,Y 256.7,Z 301.119,A -85,B 0,C 180,E1 -18361.569,E2 -18361.569} C_VEL
LIN {X 0,Y 256.454,Z 301.151,A -85,B 0,C 180,E1 -18366.293,E2 -18366.293} C_VEL
LIN {X 0,Y 256.425,Z 301.163,A -85,B 0,C 180,E1 -18369.465,E2 -18369.465} C_VEL
LIN {X 0,Y 256.253,Z 301.182,A -85,B 0,C 180,E1 -18374.29,E2 -18374.29} C_VEL
LIN {X 0,Y 256.209,Z 301.198,A -85,B 0,C 180,E1 -18377.562,E2 -18377.562} C_VEL
LIN {X 0,Y 256.181,Z 301.2,A -85,B 0,C 180,E1 -18381.135,E2 -18381.135} C_VEL
LIN {X 0,Y 256.132,Z 301.164,A -85,B 0,C 180,E1 -18385.113,E2 -18385.113} C_VEL
LIN {X 0,Y 256.054,Z 301.208,A -85,B 0,C 180,E1 -18389.607,E2 -18389.607} C_VEL
LIN {X 0,Y 256.064,Z 301.189,A -85,B 0,C 180,E1 -18393.293,E2 -18393.293} C_VEL
LIN {X 0,Y 256.111,Z 301.182,A -85,B 0,C 180,E1 -18397.271,E2 -18397.271} C_VEL
LIN {X 0,Y 256.093,Z 301.286,A -85,B 0,C 180,E1 -18398.383,E2 -18398.383} C_VEL
LIN {X 0,Y 258.617,Z 308.881,A -85,B 0,C 180,E1 -18401.83,E2 -18401.83} C_VEL
LIN {X 0,Y 261.959,Z 314.088,A -85,B 0,C 180,E1 -18402.839,E2 -18402.839} C_VEL
LIN {X 0,Y 269.434,Z 326.509,A -85,B 0,C 180,E1 -18404.971,E2 -18404.971} C_VEL
LIN {X 0,Y 276.851,Z 339.831,A -85,B 0,C 180,E1 -18406.938,E2 -18406.938} C_VEL
LIN {X 0,Y 284.066,Z 354.426,A -85,B 0,C 180,E1 -18408.753,E2 -18408.753} C_VEL
LIN {X 0,Y 290.351,Z 369.213,A -85,B 0,C 180,E1 -18410.288,E2 -18410.288} C_VEL
LIN {X 0,Y 291.1,Z 374.845,A -85,B 0,C 180,E1 -18410.585,E2 -18410.585} C_VEL
LIN {X 0,Y 286.547,Z 473.581,A -85,B 0,C 180,E1 -18412.956,E2 -18412.956} C_VEL
LIN {X 0,Y 285.18,Z 489.226,A -85,B 0,C 180,E1 -18413.521,E2 -18413.521} C_VEL
LIN {X 0,Y 283.125,Z 504.262,A -85,B 0,C 180,E1 -18414.315,E2 -18414.315} C_VEL
LIN {X 0,Y 280.751,Z 517.847,A -85,B 0,C 180,E1 -18415.286,E2 -18415.286} C_VEL
LIN {X 0,Y 277.688,Z 532.661,A -85,B 0,C 180,E1 -18416.673,E2 -18416.673} C_VEL
LIN {X 0,Y 274.391,Z 546.456,A -85,B 0,C 180,E1 -18418.328,E2 -18418.328} C_VEL
LIN {X 0,Y 270.846,Z 559.339,A -85,B 0,C 180,E1 -18420.248,E2 -18420.248} C_VEL
LIN {X 0,Y 267.67,Z 570.134,A -85,B 0,C 180,E1 -18422.223,E2 -18422.223} C_VEL
LIN {X 0,Y 264.39,Z 581.025,A -85,B 0,C 180,E1 -18424.66,E2 -18424.66} C_VEL
LIN {X 0,Y 261.345,Z 591.172,A -85,B 0,C 180,E1 -18427.468,E2 -18427.468} C_VEL
LIN {X 0,Y 258.858,Z 599.125,A -85,B 0,C 180,E1 -18430.162,E2 -18430.162} C_VEL
LIN {X 0,Y 256.634,Z 606.846,A -85,B 0,C 180,E1 -18433.432,E2 -18433.432} C_VEL
LIN {X 0,Y 255.32,Z 612.476,A -85,B 0,C 180,E1 -18436.47,E2 -18436.47} C_VEL
LIN {X 0,Y 254.553,Z 615.995,A -85,B 0,C 180,E1 -18438.857,E2 -18438.857} C_VEL
LIN {X 0,Y 254.112,Z 619.562,A -85,B 0,C 180,E1 -18442.052,E2 -18442.052} C_VEL
LIN {X 0,Y 253.992,Z 621.912,A -85,B 0,C 180,E1 -18445.239,E2 -18445.239} C_VEL
LIN {X 0,Y 254.075,Z 623.098,A -85,B 0,C 180,E1 -18448.416,E2 -18448.416} C_VEL
LIN {X 0,Y 254.075,Z 623.094,A -85,B 0,C 180,E1 -18451.586,E2 -18451.586} C_VEL
LIN {X 0,Y 254.021,Z 621.708,A -85,B 0,C 180,E1 -18455.12,E2 -18455.12} C_VEL
LIN {X 0,Y 254.101,Z 619.526,A -85,B 0,C 180,E1 -18457.95,E2 -18457.95} C_VEL
LIN {X 0,Y 254.548,Z 615.951,A -85,B 0,C 180,E1 -18461.144,E2 -18461.144} C_VEL
LIN {X 0,Y 255.599,Z 611.085,A -85,B 0,C 180,E1 -18464.328,E2 -18464.328} C_VEL
LIN {X 0,Y 257.215,Z 604.797,A -85,B 0,C 180,E1 -18467.492,E2 -18467.492} C_VEL
LIN {X 0,Y 259.475,Z 596.914,A -85,B 0,C 180,E1 -18470.617,E2 -18470.617} C_VEL
LIN {X 0,Y 262.142,Z 588.548,A -85,B 0,C 180,E1 -18473.295,E2 -18473.295} C_VEL
LIN {X 0,Y 265.061,Z 578.793,A -85,B 0,C 180,E1 -18475.86,E2 -18475.86} C_VEL
LIN {X 0,Y 268.24,Z 568.181,A -85,B 0,C 180,E1 -18478.14,E2 -18478.14} C_VEL
LIN {X 0,Y 271.762,Z 555.924,A -85,B 0,C 180,E1 -18480.285,E2 -18480.285} C_VEL
LIN {X 0,Y 275.402,Z 542.282,A -85,B 0,C 180,E1 -18482.19,E2 -18482.19} C_VEL
LIN {X 0,Y 278.529,Z 528.606,A -85,B 0,C 180,E1 -18483.72,E2 -18483.72} C_VEL
LIN {X 0,Y 281.293,Z 514.438,A -85,B 0,C 180,E1 -18484.967,E2 -18484.967} C_VEL
LIN {X 0,Y 283.74,Z 499.856,A -85,B 0,C 180,E1 -18485.926,E2 -18485.926} C_VEL
LIN {X 0,Y 285.571,Z 484.872,A -85,B 0,C 180,E1 -18486.642,E2 -18486.642} C_VEL
LIN {X 0,Y 286.684,Z 469.42,A -85,B 0,C 180,E1 -18487.135,E2 -18487.135} C_VEL
LIN {X 0,Y 291.001,Z 374.792,A -85,B 0,C 180,E1 -18489.391,E2 -18489.391} C_VEL
LIN {X 0,Y 289.973,Z 368.391,A -85,B 0,C 180,E1 -18489.757,E2 -18489.757} C_VEL
LIN {X 0,Y 282.766,Z 351.752,A -85,B 0,C 180,E1 -18491.518,E2 -18491.518} C_VEL
LIN {X 0,Y 274.593,Z 335.652,A -85,B 0,C 180,E1 -18493.595,E2 -18493.595} C_VEL
LIN {X 0,Y 267.682,Z 323.519,A -85,B 0,C 180,E1 -18495.456,E2 -18495.456} C_VEL
LIN {X 0,Y 264.326,Z 318.126,A -85,B 0,C 180,E1 -18496.399,E2 -18496.399} C_VEL
LIN {X 0,Y 261.154,Z 313.032,A -85,B 0,C 180,E1 -18497.328,E2 -18497.328} C_VEL
LIN {X 0,Y 258.528,Z 308.674,A -85,B 0,C 180,E1 -18498.156,E2 -18498.156} C_VEL
LIN {X 0,Y 256.098,Z 301.204,A -85,B 0,C 180,E1 -18501.617,E2 -18501.617} C_VEL
LIN {X 0,Y 256.108,Z 301.201,A -85,B 0,C 180,E1 -18505.413,E2 -18505.413} C_VEL
LIN {X 0,Y 256.086,Z 301.204,A -85,B 0,C 180,E1 -18508.572,E2 -18508.572} C_VEL
LIN {X 0,Y 256.097,Z 301.206,A -85,B 0,C 180,E1 -18512.191,E2 -18512.191} C_VEL
LIN {X 0,Y 256.138,Z 301.202,A -85,B 0,C 180,E1 -18515.696,E2 -18515.696} C_VEL
LIN {X 0,Y 256.167,Z 301.2,A -85,B 0,C 180,E1 -18519.105,E2 -18519.105} C_VEL
LIN {X 0,Y 256.305,Z 301.176,A -85,B 0,C 180,E1 -18524.086,E2 -18524.086} C_VEL
LIN {X 0,Y 256.298,Z 301.184,A -85,B 0,C 180,E1 -18527.328,E2 -18527.328} C_VEL
LIN {X 0,Y 256.439,Z 301.168,A -85,B 0,C 180,E1 -18530.623,E2 -18530.623} C_VEL
LIN {X 0,Y 256.459,Z 301.155,A -85,B 0,C 180,E1 -18533.707,E2 -18533.707} C_VEL
LIN {X 0,Y 256.704,Z 301.129,A -85,B 0,C 180,E1 -18538.431,E2 -18538.431} C_VEL
LIN {X 0,Y 256.702,Z 301.123,A -85,B 0,C 180,E1 -18541.569,E2 -18541.569} C_VEL
LIN {X 0,Y 256.452,Z 301.154,A -85,B 0,C 180,E1 -18546.57,E2 -18546.57} C_VEL
LIN {X 0,Y 256.406,Z 301.164,A -85,B 0,C 180,E1 -18549.466,E2 -18549.466} C_VEL
LIN {X 0,Y 256.211,Z 301.185,A -85,B 0,C 180,E1 -18554.293,E2 -18554.293} C_VEL
LIN {X 0,Y 256.151,Z 301.2,A -85,B 0,C 180,E1 -18557.566,E2 -18557.566} C_VEL
LIN {X 0,Y 256.123,Z 301.208,A -85,B 0,C 180,E1 -18561.097,E2 -18561.097} C_VEL
LIN {X 0,Y 256.088,Z 301.21,A -85,B 0,C 180,E1 -18565.088,E2 -18565.088} C_VEL
LIN {X 0,Y 256.079,Z 301.178,A -85,B 0,C 180,E1 -18568.569,E2 -18568.569} C_VEL
LIN {X 0,Y 256.074,Z 301.212,A -85,B 0,C 180,E1 -18571.699,E2 -18571.699} C_VEL
LIN {X 0,Y 256.082,Z 301.207,A -85,B 0,C 180,E1 -18575.193,E2 -18575.193} C_VEL
LIN {X 0,Y 256.067,Z 301.206,A -85,B 0,C 180,E1 -18579.143,E2 -18579.143} C_VEL
LIN {X 0,Y 256.035,Z 301.229,A -85,B 0,C 180,E1 -18581.518,E2 -18581.518} C_VEL
LIN {X 0,Y 256.938,Z 303.903,A -85,B 0,C 180,E1 -18581.858,E2 -18581.858} C_VEL
LIN {X 0,Y 259.013,Z 306.155,A -85,B 0,C 180,E1 -18582.464,E2 -18582.464} C_VEL
LIN {X 0,Y 261.926,Z 310.413,A -85,B 0,C 180,E1 -18583.331,E2 -18583.331} C_VEL
LIN {X 0,Y 263.315,Z 312.341,A -85,B 0,C 180,E1 -18583.729,E2 -18583.729} C_VEL
LIN {X 0,Y 269.52,Z 321.23,A -85,B 0,C 180,E1 -18585.433,E2 -18585.433} C_VEL
LIN {X 0,Y 276.621,Z 332.096,A -85,B 0,C 180,E1 -18587.258,E2 -18587.258} C_VEL
LIN {X 0,Y 283.559,Z 343.57,A -85,B 0,C 180,E1 -18588.933,E2 -18588.933} C_VEL
LIN {X 0,Y 288.113,Z 352.631,A -85,B 0,C 180,E1 -18590.016,E2 -18590.016} C_VEL
LIN {X 0,Y 291.54,Z 360.085,A -85,B 0,C 180,E1 -18590.818,E2 -18590.818} C_VEL
LIN {X 0,Y 286.918,Z 459.663,A -85,B 0,C 180,E1 -18593.23,E2 -18593.23} C_VEL
LIN {X 0,Y 285.5,Z 474.913,A -85,B 0,C 180,E1 -18593.846,E2 -18593.846} C_VEL
LIN {X 0,Y 283.579,Z 490.167,A -85,B 0,C 180,E1 -18594.761,E2 -18594.761} C_VEL
LIN {X 0,Y 281.262,Z 504.409,A -85,B 0,C 180,E1 -18595.905,E2 -18595.905} C_VEL
LIN {X 0,Y 278.439,Z 518.464,A -85,B 0,C 180,E1 -18597.348,E2 -18597.348} C_VEL
LIN {X 0,Y 275.224,Z 531.899,A -85,B 0,C 180,E1 -18599.075,E2 -18599.075} C_VEL
LIN {X 0,Y 271.832,Z 544.092,A -85,B 0,C 180,E1 -18601.002,E2 -18601.002} C_VEL
LIN {X 0,Y 268.613,Z 555.697,A -85,B 0,C 180,E1 -18603.301,E2 -18603.301} C_VEL
LIN {X 0,Y 265.373,Z 565.954,A -85,B 0,C 180,E1 -18605.763,E2 -18605.763} C_VEL
LIN {X 0,Y 262.444,Z 574.891,A -85,B 0,C 180,E1 -18608.394,E2 -18608.394} C_VEL
LIN {X 0,Y 259.95,Z 582.444,A -85,B 0,C 180,E1 -18611.131,E2 -18611.131} C_VEL
LIN {X 0,Y 257.924,Z 589.195,A -85,B 0,C 180,E1 -18614.187,E2 -18614.187} C_VEL
LIN {X 0,Y 256.217,Z 594.62,A -85,B 0,C 180,E1 -18617.323,E2 -18617.323} C_VEL
LIN {X 0,Y 255.136,Z 598.706,A -85,B 0,C 180,E1 -18620.486,E2 -18620.486} C_VEL
LIN {X 0,Y 254.517,Z 601.641,A -85,B 0,C 180,E1 -18623.758,E2 -18623.758} C_VEL
LIN {X 0,Y 254.236,Z 603.291,A -85,B 0,C 180,E1 -18626.83,E2 -18626.83} C_VEL
LIN {X 0,Y 254.111,Z 603.892,A -85,B 0,C 180,E1 -18629.999,E2 -18629.999} C_VEL
LIN {X 0,Y 254.235,Z 603.33,A -85,B 0,C 180,E1 -18633.169,E2 -18633.169} C_VEL
LIN {X 0,Y 254.525,Z 601.663,A -85,B 0,C 180,E1 -18636.34,E2 -18636.34} C_VEL
LIN {X 0,Y 255.131,Z 598.846,A -85,B 0,C 180,E1 -18639.513,E2 -18639.513} C_VEL
LIN {X 0,Y 256.181,Z 594.808,A -85,B 0,C 180,E1 -18642.677,E2 -18642.677} C_VEL
LIN {X 0,Y 257.847,Z 589.444,A -85,B 0,C 180,E1 -18645.816,E2 -18645.816} C_VEL
LIN {X 0,Y 259.944,Z 582.607,A -85,B 0,C 180,E1 -18648.931,E2 -18648.931} C_VEL
LIN {X 0,Y 262.755,Z 574.059,A -85,B 0,C 180,E1 -18651.99,E2 -18651.99} C_VEL
LIN {X 0,Y 265.691,Z 564.965,A -85,B 0,C 180,E1 -18654.62,E2 -18654.62} C_VEL
LIN {X 0,Y 268.627,Z 555.707,A -85,B 0,C 180,E1 -18656.823,E2 -18656.823} C_VEL
LIN {X 0,Y 271.763,Z 544.68,A -85,B 0,C 180,E1 -18659.004,E2 -18659.004} C_VEL
LIN {X 0,Y 275.127,Z 532.601,A -85,B 0,C 180,E1 -18660.936,E2 -18660.936} C_VEL
LIN {X 0,Y 278.001,Z 520.752,A -85,B 0,C 180,E1 -18662.493,E2 -18662.493} C_VEL
LIN {X 0,Y 280.68,Z 507.728,A -85,B 0,C 180,E1 -18663.899,E2 -18663.899} C_VEL
LIN {X 0,Y 283.024,Z 494.333,A -85,B 0,C 180,E1 -18665.045,E2 -18665.045} C_VEL
LIN {X 0,Y 285.067,Z 479.707,A -85,B 0,C 180,E1 -18666.003,E2 -18666.003} C_VEL
LIN {X 0,Y 286.56,Z 464.686,A -85,B 0,C 180,E1 -18666.712,E2 -18666.712} C_VEL
LIN {X 0,Y 287.712,Z 447.679,A -85,B 0,C 180,E1 -18667.197,E2 -18667.197} C_VEL
LIN {X 0,Y 291.596,Z 360.193,A -85,B 0,C 180,E1 -18669.301,E2 -18669.301} C_VEL
LIN {X 0,Y 285.116,Z 346.319,A -85,B 0,C 180,E1 -18670.838,E2 -18670.838} C_VEL
LIN {X 0,Y 277.504,Z 333.387,A -85,B 0,C 180,E1 -18672.669,E2 -18672.669} C_VEL
LIN {X 0,Y 270.15,Z 322.109,A -85,B 0,C 180,E1 -18674.549,E2 -18674.549} C_VEL
LIN {X 0,Y 265.011,Z 314.659,A -85,B 0,C 180,E1 -18675.948,E2 -18675.948} C_VEL
LIN {X 0,Y 262.102,Z 310.552,A -85,B 0,C 180,E1 -18676.776,E2 -18676.776} C_VEL
LIN {X 0,Y 259.813,Z 307.375,A -85,B 0,C 180,E1 -18677.448,E2 -18677.448} C_VEL
LIN {X 0,Y 259.173,Z 306.239,A -85,B 0,C 180,E1 -18677.65,E2 -18677.65} C_VEL
LIN {X 0,Y 256.953,Z 303.916,A -85,B 0,C 180,E1 -18678.297,E2 -18678.297} C_VEL
LIN {X 0,Y 256.012,Z 301.195,A -85,B 0,C 180,E1 -18678.684,E2 -18678.684} C_VEL
LIN {X 0,Y 256.097,Z 301.177,A -85,B 0,C 180,E1 -18682.861,E2 -18682.861} C_VEL
LIN {X 0,Y 256.063,Z 301.214,A -85,B 0,C 180,E1 -18686.706,E2 -18686.706} C_VEL
LIN {X 0,Y 256.038,Z 301.217,A -85,B 0,C 180,E1 -18690.391,E2 -18690.391} C_VEL
LIN {X 0,Y 256.041,Z 301.209,A -85,B 0,C 180,E1 -18693.385,E2 -18693.385} C_VEL
LIN {X 0,Y 255.405,Z 301.297,A -85,B 0,C 180,E1 -18694.698,E2 -18694.698} C_VEL
LIN {X 0,Y 252.591,Z 301.652,A -85,B 0,C 180,E1 -18696.838,E2 -18696.838} C_VEL
LIN {X 0,Y 250.177,Z 301.948,A -85,B 0,C 180,E1 -18698.579,E2 -18698.579} C_VEL
LIN {X 0,Y 249.126,Z 302.072,A -85,B 0,C 180,E1 -18699.929,E2 -18699.929} C_VEL
LIN {X 0,Y 249.033,Z 302.078,A -85,B 0,C 180,E1 -18700.387,E2 -18700.387} C_VEL
LIN {X 0,Y 249.156,Z 302.075,A -85,B 0,C 180,E1 -18703.616,E2 -18703.616} C_VEL
LIN {X 0,Y 249.227,Z 302.066,A -85,B 0,C 180,E1 -18708.615,E2 -18708.615} C_VEL
LIN {X 0,Y 249.415,Z 302.031,A -85,B 0,C 180,E1 -18711.901,E2 -18711.901} C_VEL
LIN {X 0,Y 249.266,Z 302.048,A -85,B 0,C 180,E1 -18715.148,E2 -18715.148} C_VEL
LIN {X 0,Y 249.659,Z 302.013,A -85,B 0,C 180,E1 -18718.387,E2 -18718.387} C_VEL
LIN {X 0,Y 249.66,Z 301.996,A -85,B 0,C 180,E1 -18721.613,E2 -18721.613} C_VEL
LIN {X 0,Y 249.428,Z 302.026,A -85,B 0,C 180,E1 -18726.471,E2 -18726.471} C_VEL
LIN {X 0,Y 249.341,Z 302.042,A -85,B 0,C 180,E1 -18729.736,E2 -18729.736} C_VEL
LIN {X 0,Y 249.204,Z 302.057,A -85,B 0,C 180,E1 -18734.703,E2 -18734.703} C_VEL
LIN {X 0,Y 249.138,Z 302.075,A -85,B 0,C 180,E1 -18738.077,E2 -18738.077} C_VEL
LIN {X 0,Y 249.095,Z 302.084,A -85,B 0,C 180,E1 -18741.517,E2 -18741.517} C_VEL
LIN {X 0,Y 249.084,Z 302.042,A -85,B 0,C 180,E1 -18745.461,E2 -18745.461} C_VEL
LIN {X 0,Y 249.037,Z 302.09,A -85,B 0,C 180,E1 -18748.975,E2 -18748.975} C_VEL
LIN {X 0,Y 249.025,Z 302.057,A -85,B 0,C 180,E1 -18752.426,E2 -18752.426} C_VEL
LIN {X 0,Y 249.074,Z 302.142,A -85,B 0,C 180,E1 -18756.834,E2 -18756.834} C_VEL
LIN {X 0,Y 251.104,Z 308.414,A -85,B 0,C 180,E1 -18759.874,E2 -18759.874} C_VEL
LIN {X 0,Y 254.308,Z 313.329,A -85,B 0,C 180,E1 -18760.931,E2 -18760.931} C_VEL
LIN {X 0,Y 259.444,Z 321.5,A -85,B 0,C 180,E1 -18762.538,E2 -18762.538} C_VEL
LIN {X 0,Y 265.218,Z 331.053,A -85,B 0,C 180,E1 -18764.232,E2 -18764.232} C_VEL
LIN {X 0,Y 272.332,Z 343.989,A -85,B 0,C 180,E1 -18766.199,E2 -18766.199} C_VEL
LIN {X 0,Y 278.953,Z 357.606,A -85,B 0,C 180,E1 -18767.941,E2 -18767.941} C_VEL
LIN {X 0,Y 285.068,Z 372.028,A -85,B 0,C 180,E1 -18769.499,E2 -18769.499} C_VEL
LIN {X 0,Y 285.536,Z 376.738,A -85,B 0,C 180,E1 -18769.731,E2 -18769.731} C_VEL
LIN {X 0,Y 281.409,Z 463.392,A -85,B 0,C 180,E1 -18771.822,E2 -18771.822} C_VEL
LIN {X 0,Y 280.307,Z 480.967,A -85,B 0,C 180,E1 -18772.329,E2 -18772.329} C_VEL
LIN {X 0,Y 278.585,Z 496.352,A -85,B 0,C 180,E1 -18773.022,E2 -18773.022} C_VEL
LIN {X 0,Y 276.135,Z 511.204,A -85,B 0,C 180,E1 -18773.946,E2 -18773.946} C_VEL
LIN {X 0,Y 273.416,Z 525.136,A -85,B 0,C 180,E1 -18775.116,E2 -18775.116} C_VEL
LIN {X 0,Y 270.536,Z 537.76,A -85,B 0,C 180,E1 -18776.459,E2 -18776.459} C_VEL
LIN {X 0,Y 266.959,Z 551.167,A -85,B 0,C 180,E1 -18778.23,E2 -18778.23} C_VEL
LIN {X 0,Y 263.767,Z 562.236,A -85,B 0,C 180,E1 -18780.028,E2 -18780.028} C_VEL
LIN {X 0,Y 260.249,Z 573.427,A -85,B 0,C 180,E1 -18782.237,E2 -18782.237} C_VEL
LIN {X 0,Y 257.322,Z 582.695,A -85,B 0,C 180,E1 -18784.476,E2 -18784.476} C_VEL
LIN {X 0,Y 254.321,Z 592.143,A -85,B 0,C 180,E1 -18787.24,E2 -18787.24} C_VEL
LIN {X 0,Y 251.498,Z 600.891,A -85,B 0,C 180,E1 -18790.408,E2 -18790.408} C_VEL
LIN {X 0,Y 249.403,Z 607.923,A -85,B 0,C 180,E1 -18793.634,E2 -18793.634} C_VEL
LIN {X 0,Y 248.049,Z 613.465,A -85,B 0,C 180,E1 -18796.9,E2 -18796.9} C_VEL
LIN {X 0,Y 247.224,Z 617.662,A -85,B 0,C 180,E1 -18800.18,E2 -18800.18} C_VEL
LIN {X 0,Y 246.952,Z 620.615,A -85,B 0,C 180,E1 -18803.464,E2 -18803.464} C_VEL
LIN {X 0,Y 246.912,Z 622.378,A -85,B 0,C 180,E1 -18806.737,E2 -18806.737} C_VEL
